// TIA Portal V20 export
FUNCTION_BLOCK "System_To_Moving_Pallets"   // FB15, LAD
{ S7_Optimized_Access := 'TRUE' }
// stored: MemoryReserve 100, SetENOAutomatically false
   VAR
      iCenterTippler : Bool;
      oCeterTippler : Bool;
      Reset_Centering_Tippler : Bool;
      ST13_ST14 { S7_SetPoint := 'True'} : "Pallet_Transport_Row_4";
      ST12_ST13 { S7_SetPoint := 'True'} : "Pallet_Transport_Row_4";
      ST11_ST12 { S7_SetPoint := 'True'} : "Pallet_Transport_Row_4";
      ST10_ST11 { S7_SetPoint := 'True'} : "Pallet_Transport_Row_4";
      ST09_ST10 { S7_SetPoint := 'True'} : "Pallet_Transport_Row_4";
      ST08_ST09 { S7_SetPoint := 'True'} : "Pallet_Transport_Row_4";
      ST07_ST08 { S7_SetPoint := 'True'} : "Pallet_Transport_Row_4";
      ST06_ST07 { S7_SetPoint := 'True'} : "Pallet_Transport_Row_4";
      ST05_ST06 { S7_SetPoint := 'True'} : "Pallet_Transport_Row_4";
      ST04_ST05 { S7_SetPoint := 'True'} : "Pallet_Transport_Row_4";
      ST01_ST02 { S7_SetPoint := 'True'} : "Pallet_Transport_Row_1_2";
      ST02_ST01 { S7_SetPoint := 'True'} : "Pallet_Transport_Row_1_2";
      ST38_ST01 { S7_SetPoint := 'True'} : "Pallet_Transport_Row_1_2";
      ST01_ST38 { S7_SetPoint := 'True'} : "Pallet_Transport_Row_1_2";
      ST34_ST35 { S7_SetPoint := 'True'} : "Pallet_Transport_Row_1_2";
      ST35_ST34 { S7_SetPoint := 'True'} : "Pallet_Transport_Row_1_2";
      ST33_ST34 { S7_SetPoint := 'True'} : "Pallet_Transport_Row_1_2";
      ST34_ST33 { S7_SetPoint := 'True'} : "Pallet_Transport_Row_1_2";
      ST32_ST33 { S7_SetPoint := 'True'} : "Pallet_Transport_Row_1_2";
      ST36_ST38 { S7_SetPoint := 'True'} : "Pallet_Transport_Row_1_2";
      ST38_ST36 { S7_SetPoint := 'True'} : "Pallet_Transport_Row_1_2";
      ST37_ST36 { S7_SetPoint := 'True'} : "Pallet_Transport_Row_1_2";
      ST18_ST37 { S7_SetPoint := 'True'} : "Pallet_Transport_Row_1_2";
      ST19_ST18 { S7_SetPoint := 'True'} : "Pallet_Transport_Row_1_2";
      ST20_ST19 { S7_SetPoint := 'True'} : "Pallet_Transport_Row_1_2";
      ST21_ST20 { S7_SetPoint := 'True'} : "Pallet_Transport_Row_1_2";
      ST22_ST21 { S7_SetPoint := 'True'} : "Pallet_Transport_Row_1_2";
      ST23_ST22 { S7_SetPoint := 'True'} : "Pallet_Transport_Row_1_2";
      ST24_ST23 { S7_SetPoint := 'True'} : "Pallet_Transport_Row_1_2";
      Centering_Perform : Array[7..13, 1..3] of Bool;
      Centering_Status { S7_SetPoint := 'True'} : Array[7..13, 1..3] of Bool;
      ST31_ST32 { S7_SetPoint := 'True'} : "Pallet_Transport_Row_1_2";
      ST30_ST31 { S7_SetPoint := 'True'} : "Pallet_Transport_Row_1_2";
      ST29_ST30 { S7_SetPoint := 'True'} : "Pallet_Transport_Row_1_2";
      ST28_ST29 { S7_SetPoint := 'True'} : "Pallet_Transport_Row_1_2";
      TON_Reset_Drives { S7_SetPoint := 'True'} : TON_TIME;
      TP_Reset_Drives { S7_SetPoint := 'True'} : TP_TIME;
      Reset_Drives_Var { S7_SetPoint := 'True'} : Bool;
      ST27_ST28 { S7_SetPoint := 'True'} : "Pallet_Transport_Row_1_2";
      ST26_ST27 { S7_SetPoint := 'True'} : "Pallet_Transport_Row_1_2";
      ST25_ST26 { S7_SetPoint := 'True'} : "Pallet_Transport_Row_1_2";
      tComm_W1 { S7_SetPoint := 'True'} : TON_TIME;
      tComm_W2 { S7_SetPoint := 'True'} : TON_TIME;
      tComm_W4 { S7_SetPoint := 'True'} : TON_TIME;
   END_VAR
   VAR_TEMP
      i : Int;
   END_VAR
BEGIN

REGION Network 1: Initialisation of pallets status
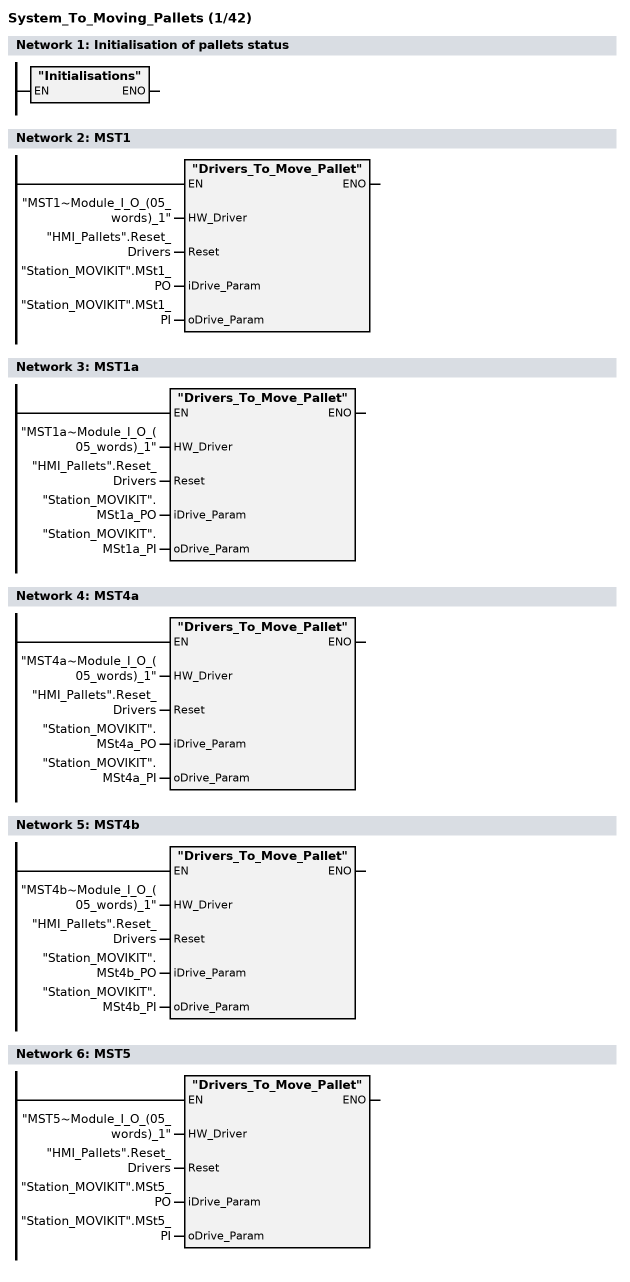
   RUNG wire#powerrail
      "Initialisations"()
   END_RUNG
   // the same network as SCL:
   "Initialisations"();
END_REGION

REGION Network 2: MST1
   RUNG wire#powerrail
      "Drivers_To_Move_Pallet"(HW_Driver := "MST1~Module_I_O_(05_words)_1", Reset := "HMI_Pallets".Reset_Drivers, iDrive_Param := "Station_MOVIKIT".MSt1_PO, oDrive_Param := "Station_MOVIKIT".MSt1_PI)
   END_RUNG
   // the same network as SCL:
   "Drivers_To_Move_Pallet"(HW_Driver := "MST1~Module_I_O_(05_words)_1",
                           Reset := "HMI_Pallets".Reset_Drivers,
                           iDrive_Param := "Station_MOVIKIT".MSt1_PO,
                           oDrive_Param := "Station_MOVIKIT".MSt1_PI);
END_REGION

REGION Network 3: MST1a
   RUNG wire#powerrail
      "Drivers_To_Move_Pallet"(HW_Driver := "MST1a~Module_I_O_(05_words)_1", Reset := "HMI_Pallets".Reset_Drivers, iDrive_Param := "Station_MOVIKIT".MSt1a_PO, oDrive_Param := "Station_MOVIKIT".MSt1a_PI)
   END_RUNG
   // the same network as SCL:
   "Drivers_To_Move_Pallet"(HW_Driver := "MST1a~Module_I_O_(05_words)_1",
                           Reset := "HMI_Pallets".Reset_Drivers,
                           iDrive_Param := "Station_MOVIKIT".MSt1a_PO,
                           oDrive_Param := "Station_MOVIKIT".MSt1a_PI);
END_REGION

REGION Network 4: MST4a
   RUNG wire#powerrail
      "Drivers_To_Move_Pallet"(HW_Driver := "MST4a~Module_I_O_(05_words)_1", Reset := "HMI_Pallets".Reset_Drivers, iDrive_Param := "Station_MOVIKIT".MSt4a_PO, oDrive_Param := "Station_MOVIKIT".MSt4a_PI)
   END_RUNG
   // the same network as SCL:
   "Drivers_To_Move_Pallet"(HW_Driver := "MST4a~Module_I_O_(05_words)_1",
                           Reset := "HMI_Pallets".Reset_Drivers,
                           iDrive_Param := "Station_MOVIKIT".MSt4a_PO,
                           oDrive_Param := "Station_MOVIKIT".MSt4a_PI);
END_REGION

REGION Network 5: MST4b
   RUNG wire#powerrail
      "Drivers_To_Move_Pallet"(HW_Driver := "MST4b~Module_I_O_(05_words)_1", Reset := "HMI_Pallets".Reset_Drivers, iDrive_Param := "Station_MOVIKIT".MSt4b_PO, oDrive_Param := "Station_MOVIKIT".MSt4b_PI)
   END_RUNG
   // the same network as SCL:
   "Drivers_To_Move_Pallet"(HW_Driver := "MST4b~Module_I_O_(05_words)_1",
                           Reset := "HMI_Pallets".Reset_Drivers,
                           iDrive_Param := "Station_MOVIKIT".MSt4b_PO,
                           oDrive_Param := "Station_MOVIKIT".MSt4b_PI);
END_REGION

REGION Network 6: MST5
   RUNG wire#powerrail
      "Drivers_To_Move_Pallet"(HW_Driver := "MST5~Module_I_O_(05_words)_1", Reset := "HMI_Pallets".Reset_Drivers, iDrive_Param := "Station_MOVIKIT".MSt5_PO, oDrive_Param := "Station_MOVIKIT".MSt5_PI)
   END_RUNG
   // the same network as SCL:
   "Drivers_To_Move_Pallet"(HW_Driver := "MST5~Module_I_O_(05_words)_1",
                           Reset := "HMI_Pallets".Reset_Drivers,
                           iDrive_Param := "Station_MOVIKIT".MSt5_PO,
                           oDrive_Param := "Station_MOVIKIT".MSt5_PI);
END_REGION

REGION Network 7: MST6a
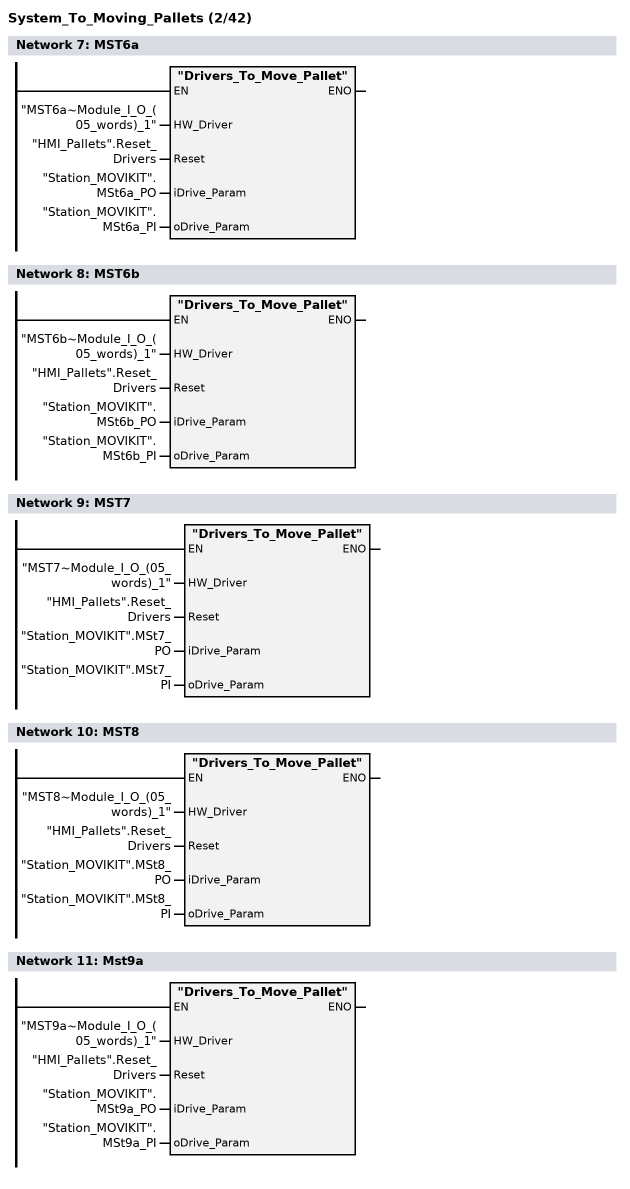
   RUNG wire#powerrail
      "Drivers_To_Move_Pallet"(HW_Driver := "MST6a~Module_I_O_(05_words)_1", Reset := "HMI_Pallets".Reset_Drivers, iDrive_Param := "Station_MOVIKIT".MSt6a_PO, oDrive_Param := "Station_MOVIKIT".MSt6a_PI)
   END_RUNG
   // the same network as SCL:
   "Drivers_To_Move_Pallet"(HW_Driver := "MST6a~Module_I_O_(05_words)_1",
                           Reset := "HMI_Pallets".Reset_Drivers,
                           iDrive_Param := "Station_MOVIKIT".MSt6a_PO,
                           oDrive_Param := "Station_MOVIKIT".MSt6a_PI);
END_REGION

REGION Network 8: MST6b
   RUNG wire#powerrail
      "Drivers_To_Move_Pallet"(HW_Driver := "MST6b~Module_I_O_(05_words)_1", Reset := "HMI_Pallets".Reset_Drivers, iDrive_Param := "Station_MOVIKIT".MSt6b_PO, oDrive_Param := "Station_MOVIKIT".MSt6b_PI)
   END_RUNG
   // the same network as SCL:
   "Drivers_To_Move_Pallet"(HW_Driver := "MST6b~Module_I_O_(05_words)_1",
                           Reset := "HMI_Pallets".Reset_Drivers,
                           iDrive_Param := "Station_MOVIKIT".MSt6b_PO,
                           oDrive_Param := "Station_MOVIKIT".MSt6b_PI);
END_REGION

REGION Network 9: MST7
   RUNG wire#powerrail
      "Drivers_To_Move_Pallet"(HW_Driver := "MST7~Module_I_O_(05_words)_1", Reset := "HMI_Pallets".Reset_Drivers, iDrive_Param := "Station_MOVIKIT".MSt7_PO, oDrive_Param := "Station_MOVIKIT".MSt7_PI)
   END_RUNG
   // the same network as SCL:
   "Drivers_To_Move_Pallet"(HW_Driver := "MST7~Module_I_O_(05_words)_1",
                           Reset := "HMI_Pallets".Reset_Drivers,
                           iDrive_Param := "Station_MOVIKIT".MSt7_PO,
                           oDrive_Param := "Station_MOVIKIT".MSt7_PI);
END_REGION

REGION Network 10: MST8
   RUNG wire#powerrail
      "Drivers_To_Move_Pallet"(HW_Driver := "MST8~Module_I_O_(05_words)_1", Reset := "HMI_Pallets".Reset_Drivers, iDrive_Param := "Station_MOVIKIT".MSt8_PO, oDrive_Param := "Station_MOVIKIT".MSt8_PI)
   END_RUNG
   // the same network as SCL:
   "Drivers_To_Move_Pallet"(HW_Driver := "MST8~Module_I_O_(05_words)_1",
                           Reset := "HMI_Pallets".Reset_Drivers,
                           iDrive_Param := "Station_MOVIKIT".MSt8_PO,
                           oDrive_Param := "Station_MOVIKIT".MSt8_PI);
END_REGION

REGION Network 11: Mst9a
   RUNG wire#powerrail
      "Drivers_To_Move_Pallet"(HW_Driver := "MST9a~Module_I_O_(05_words)_1", Reset := "HMI_Pallets".Reset_Drivers, iDrive_Param := "Station_MOVIKIT".MSt9a_PO, oDrive_Param := "Station_MOVIKIT".MSt9a_PI)
   END_RUNG
   // the same network as SCL:
   "Drivers_To_Move_Pallet"(HW_Driver := "MST9a~Module_I_O_(05_words)_1",
                           Reset := "HMI_Pallets".Reset_Drivers,
                           iDrive_Param := "Station_MOVIKIT".MSt9a_PO,
                           oDrive_Param := "Station_MOVIKIT".MSt9a_PI);
END_REGION

REGION Network 12: Mst9b
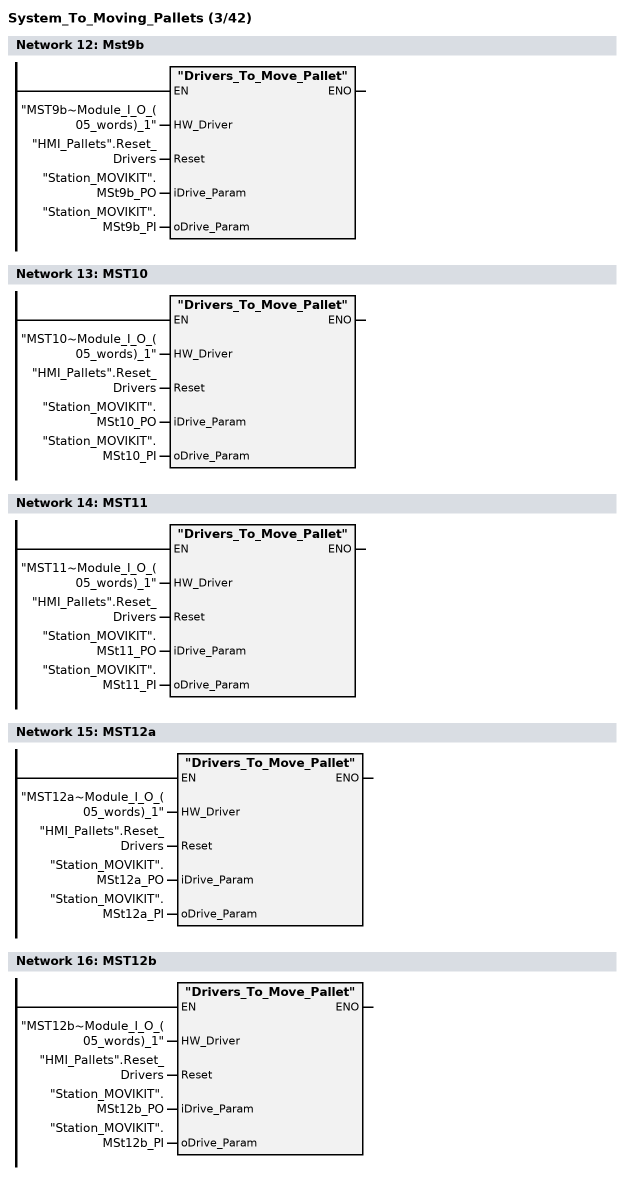
   RUNG wire#powerrail
      "Drivers_To_Move_Pallet"(HW_Driver := "MST9b~Module_I_O_(05_words)_1", Reset := "HMI_Pallets".Reset_Drivers, iDrive_Param := "Station_MOVIKIT".MSt9b_PO, oDrive_Param := "Station_MOVIKIT".MSt9b_PI)
   END_RUNG
   // the same network as SCL:
   "Drivers_To_Move_Pallet"(HW_Driver := "MST9b~Module_I_O_(05_words)_1",
                           Reset := "HMI_Pallets".Reset_Drivers,
                           iDrive_Param := "Station_MOVIKIT".MSt9b_PO,
                           oDrive_Param := "Station_MOVIKIT".MSt9b_PI);
END_REGION

REGION Network 13: MST10
   RUNG wire#powerrail
      "Drivers_To_Move_Pallet"(HW_Driver := "MST10~Module_I_O_(05_words)_1", Reset := "HMI_Pallets".Reset_Drivers, iDrive_Param := "Station_MOVIKIT".MSt10_PO, oDrive_Param := "Station_MOVIKIT".MSt10_PI)
   END_RUNG
   // the same network as SCL:
   "Drivers_To_Move_Pallet"(HW_Driver := "MST10~Module_I_O_(05_words)_1",
                           Reset := "HMI_Pallets".Reset_Drivers,
                           iDrive_Param := "Station_MOVIKIT".MSt10_PO,
                           oDrive_Param := "Station_MOVIKIT".MSt10_PI);
END_REGION

REGION Network 14: MST11
   RUNG wire#powerrail
      "Drivers_To_Move_Pallet"(HW_Driver := "MST11~Module_I_O_(05_words)_1", Reset := "HMI_Pallets".Reset_Drivers, iDrive_Param := "Station_MOVIKIT".MSt11_PO, oDrive_Param := "Station_MOVIKIT".MSt11_PI)
   END_RUNG
   // the same network as SCL:
   "Drivers_To_Move_Pallet"(HW_Driver := "MST11~Module_I_O_(05_words)_1",
                           Reset := "HMI_Pallets".Reset_Drivers,
                           iDrive_Param := "Station_MOVIKIT".MSt11_PO,
                           oDrive_Param := "Station_MOVIKIT".MSt11_PI);
END_REGION

REGION Network 15: MST12a
   RUNG wire#powerrail
      "Drivers_To_Move_Pallet"(HW_Driver := "MST12a~Module_I_O_(05_words)_1", Reset := "HMI_Pallets".Reset_Drivers, iDrive_Param := "Station_MOVIKIT".MSt12a_PO, oDrive_Param := "Station_MOVIKIT".MSt12a_PI)
   END_RUNG
   // the same network as SCL:
   "Drivers_To_Move_Pallet"(HW_Driver := "MST12a~Module_I_O_(05_words)_1",
                           Reset := "HMI_Pallets".Reset_Drivers,
                           iDrive_Param := "Station_MOVIKIT".MSt12a_PO,
                           oDrive_Param := "Station_MOVIKIT".MSt12a_PI);
END_REGION

REGION Network 16: MST12b
   RUNG wire#powerrail
      "Drivers_To_Move_Pallet"(HW_Driver := "MST12b~Module_I_O_(05_words)_1", Reset := "HMI_Pallets".Reset_Drivers, iDrive_Param := "Station_MOVIKIT".MSt12b_PO, oDrive_Param := "Station_MOVIKIT".MSt12b_PI)
   END_RUNG
   // the same network as SCL:
   "Drivers_To_Move_Pallet"(HW_Driver := "MST12b~Module_I_O_(05_words)_1",
                           Reset := "HMI_Pallets".Reset_Drivers,
                           iDrive_Param := "Station_MOVIKIT".MSt12b_PO,
                           oDrive_Param := "Station_MOVIKIT".MSt12b_PI);
END_REGION

REGION Network 17: MST13
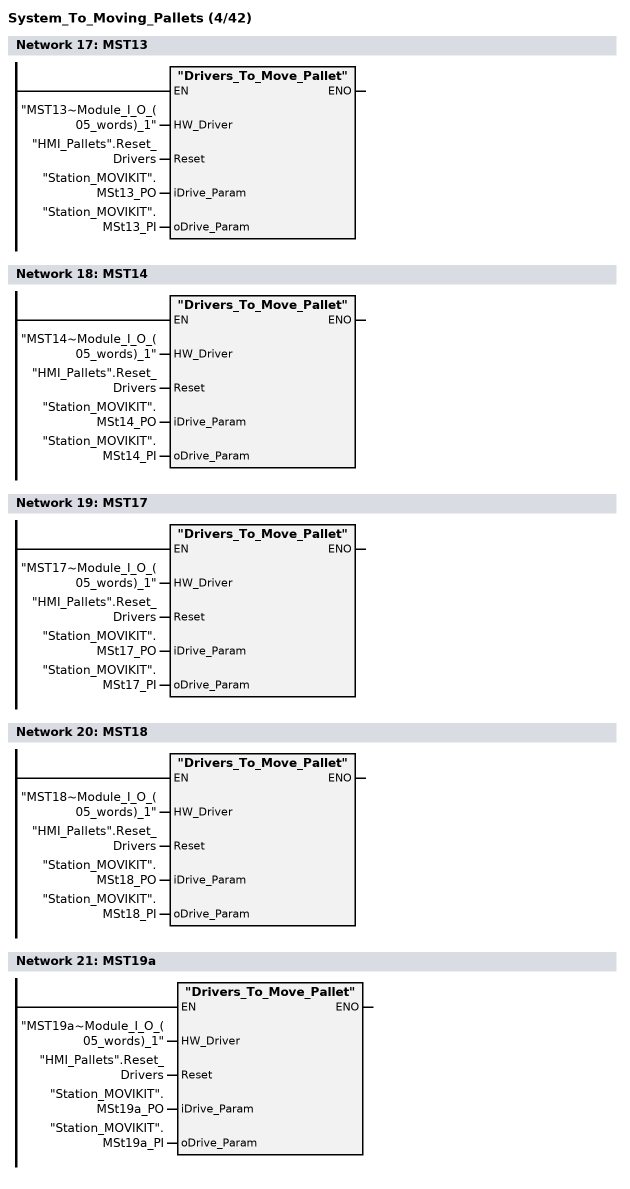
   RUNG wire#powerrail
      "Drivers_To_Move_Pallet"(HW_Driver := "MST13~Module_I_O_(05_words)_1", Reset := "HMI_Pallets".Reset_Drivers, iDrive_Param := "Station_MOVIKIT".MSt13_PO, oDrive_Param := "Station_MOVIKIT".MSt13_PI)
   END_RUNG
   // the same network as SCL:
   "Drivers_To_Move_Pallet"(HW_Driver := "MST13~Module_I_O_(05_words)_1",
                           Reset := "HMI_Pallets".Reset_Drivers,
                           iDrive_Param := "Station_MOVIKIT".MSt13_PO,
                           oDrive_Param := "Station_MOVIKIT".MSt13_PI);
END_REGION

REGION Network 18: MST14
   RUNG wire#powerrail
      "Drivers_To_Move_Pallet"(HW_Driver := "MST14~Module_I_O_(05_words)_1", Reset := "HMI_Pallets".Reset_Drivers, iDrive_Param := "Station_MOVIKIT".MSt14_PO, oDrive_Param := "Station_MOVIKIT".MSt14_PI)
   END_RUNG
   // the same network as SCL:
   "Drivers_To_Move_Pallet"(HW_Driver := "MST14~Module_I_O_(05_words)_1",
                           Reset := "HMI_Pallets".Reset_Drivers,
                           iDrive_Param := "Station_MOVIKIT".MSt14_PO,
                           oDrive_Param := "Station_MOVIKIT".MSt14_PI);
END_REGION

REGION Network 19: MST17
   RUNG wire#powerrail
      "Drivers_To_Move_Pallet"(HW_Driver := "MST17~Module_I_O_(05_words)_1", Reset := "HMI_Pallets".Reset_Drivers, iDrive_Param := "Station_MOVIKIT".MSt17_PO, oDrive_Param := "Station_MOVIKIT".MSt17_PI)
   END_RUNG
   // the same network as SCL:
   "Drivers_To_Move_Pallet"(HW_Driver := "MST17~Module_I_O_(05_words)_1",
                           Reset := "HMI_Pallets".Reset_Drivers,
                           iDrive_Param := "Station_MOVIKIT".MSt17_PO,
                           oDrive_Param := "Station_MOVIKIT".MSt17_PI);
END_REGION

REGION Network 20: MST18
   RUNG wire#powerrail
      "Drivers_To_Move_Pallet"(HW_Driver := "MST18~Module_I_O_(05_words)_1", Reset := "HMI_Pallets".Reset_Drivers, iDrive_Param := "Station_MOVIKIT".MSt18_PO, oDrive_Param := "Station_MOVIKIT".MSt18_PI)
   END_RUNG
   // the same network as SCL:
   "Drivers_To_Move_Pallet"(HW_Driver := "MST18~Module_I_O_(05_words)_1",
                           Reset := "HMI_Pallets".Reset_Drivers,
                           iDrive_Param := "Station_MOVIKIT".MSt18_PO,
                           oDrive_Param := "Station_MOVIKIT".MSt18_PI);
END_REGION

REGION Network 21: MST19a
   RUNG wire#powerrail
      "Drivers_To_Move_Pallet"(HW_Driver := "MST19a~Module_I_O_(05_words)_1", Reset := "HMI_Pallets".Reset_Drivers, iDrive_Param := "Station_MOVIKIT".MSt19a_PO, oDrive_Param := "Station_MOVIKIT".MSt19a_PI)
   END_RUNG
   // the same network as SCL:
   "Drivers_To_Move_Pallet"(HW_Driver := "MST19a~Module_I_O_(05_words)_1",
                           Reset := "HMI_Pallets".Reset_Drivers,
                           iDrive_Param := "Station_MOVIKIT".MSt19a_PO,
                           oDrive_Param := "Station_MOVIKIT".MSt19a_PI);
END_REGION

REGION Network 22: MST19b
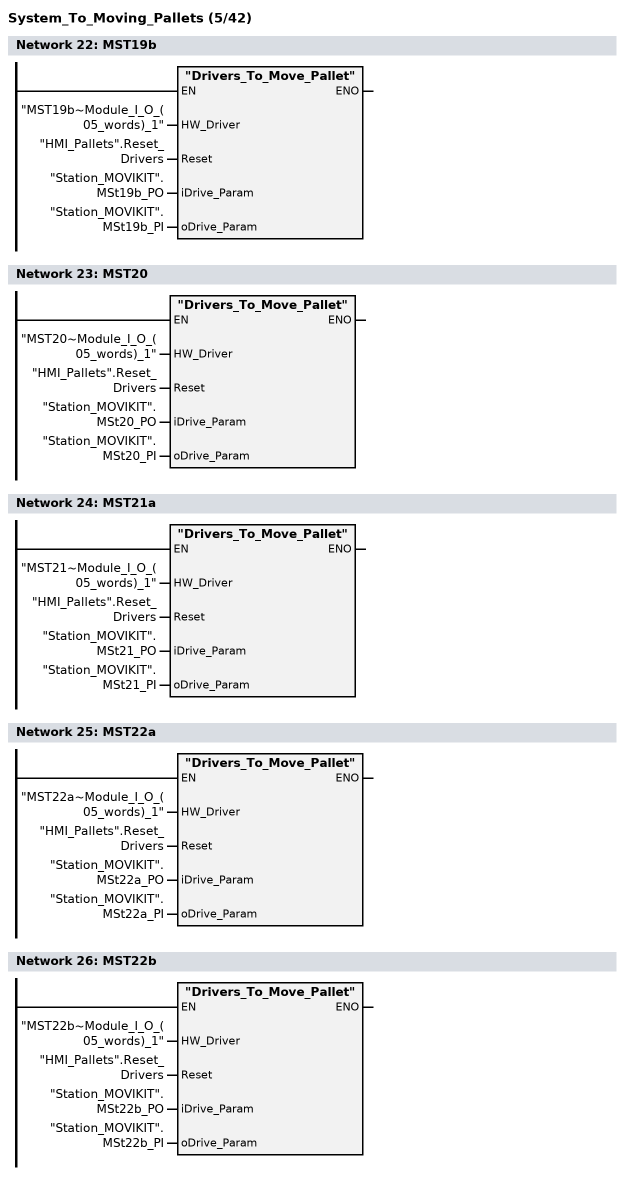
   RUNG wire#powerrail
      "Drivers_To_Move_Pallet"(HW_Driver := "MST19b~Module_I_O_(05_words)_1", Reset := "HMI_Pallets".Reset_Drivers, iDrive_Param := "Station_MOVIKIT".MSt19b_PO, oDrive_Param := "Station_MOVIKIT".MSt19b_PI)
   END_RUNG
   // the same network as SCL:
   "Drivers_To_Move_Pallet"(HW_Driver := "MST19b~Module_I_O_(05_words)_1",
                           Reset := "HMI_Pallets".Reset_Drivers,
                           iDrive_Param := "Station_MOVIKIT".MSt19b_PO,
                           oDrive_Param := "Station_MOVIKIT".MSt19b_PI);
END_REGION

REGION Network 23: MST20
   RUNG wire#powerrail
      "Drivers_To_Move_Pallet"(HW_Driver := "MST20~Module_I_O_(05_words)_1", Reset := "HMI_Pallets".Reset_Drivers, iDrive_Param := "Station_MOVIKIT".MSt20_PO, oDrive_Param := "Station_MOVIKIT".MSt20_PI)
   END_RUNG
   // the same network as SCL:
   "Drivers_To_Move_Pallet"(HW_Driver := "MST20~Module_I_O_(05_words)_1",
                           Reset := "HMI_Pallets".Reset_Drivers,
                           iDrive_Param := "Station_MOVIKIT".MSt20_PO,
                           oDrive_Param := "Station_MOVIKIT".MSt20_PI);
END_REGION

REGION Network 24: MST21a
   RUNG wire#powerrail
      "Drivers_To_Move_Pallet"(HW_Driver := "MST21~Module_I_O_(05_words)_1", Reset := "HMI_Pallets".Reset_Drivers, iDrive_Param := "Station_MOVIKIT".MSt21_PO, oDrive_Param := "Station_MOVIKIT".MSt21_PI)
   END_RUNG
   // the same network as SCL:
   "Drivers_To_Move_Pallet"(HW_Driver := "MST21~Module_I_O_(05_words)_1",
                           Reset := "HMI_Pallets".Reset_Drivers,
                           iDrive_Param := "Station_MOVIKIT".MSt21_PO,
                           oDrive_Param := "Station_MOVIKIT".MSt21_PI);
END_REGION

REGION Network 25: MST22a
   RUNG wire#powerrail
      "Drivers_To_Move_Pallet"(HW_Driver := "MST22a~Module_I_O_(05_words)_1", Reset := "HMI_Pallets".Reset_Drivers, iDrive_Param := "Station_MOVIKIT".MSt22a_PO, oDrive_Param := "Station_MOVIKIT".MSt22a_PI)
   END_RUNG
   // the same network as SCL:
   "Drivers_To_Move_Pallet"(HW_Driver := "MST22a~Module_I_O_(05_words)_1",
                           Reset := "HMI_Pallets".Reset_Drivers,
                           iDrive_Param := "Station_MOVIKIT".MSt22a_PO,
                           oDrive_Param := "Station_MOVIKIT".MSt22a_PI);
END_REGION

REGION Network 26: MST22b
   RUNG wire#powerrail
      "Drivers_To_Move_Pallet"(HW_Driver := "MST22b~Module_I_O_(05_words)_1", Reset := "HMI_Pallets".Reset_Drivers, iDrive_Param := "Station_MOVIKIT".MSt22b_PO, oDrive_Param := "Station_MOVIKIT".MSt22b_PI)
   END_RUNG
   // the same network as SCL:
   "Drivers_To_Move_Pallet"(HW_Driver := "MST22b~Module_I_O_(05_words)_1",
                           Reset := "HMI_Pallets".Reset_Drivers,
                           iDrive_Param := "Station_MOVIKIT".MSt22b_PO,
                           oDrive_Param := "Station_MOVIKIT".MSt22b_PI);
END_REGION

REGION Network 27: MST23a
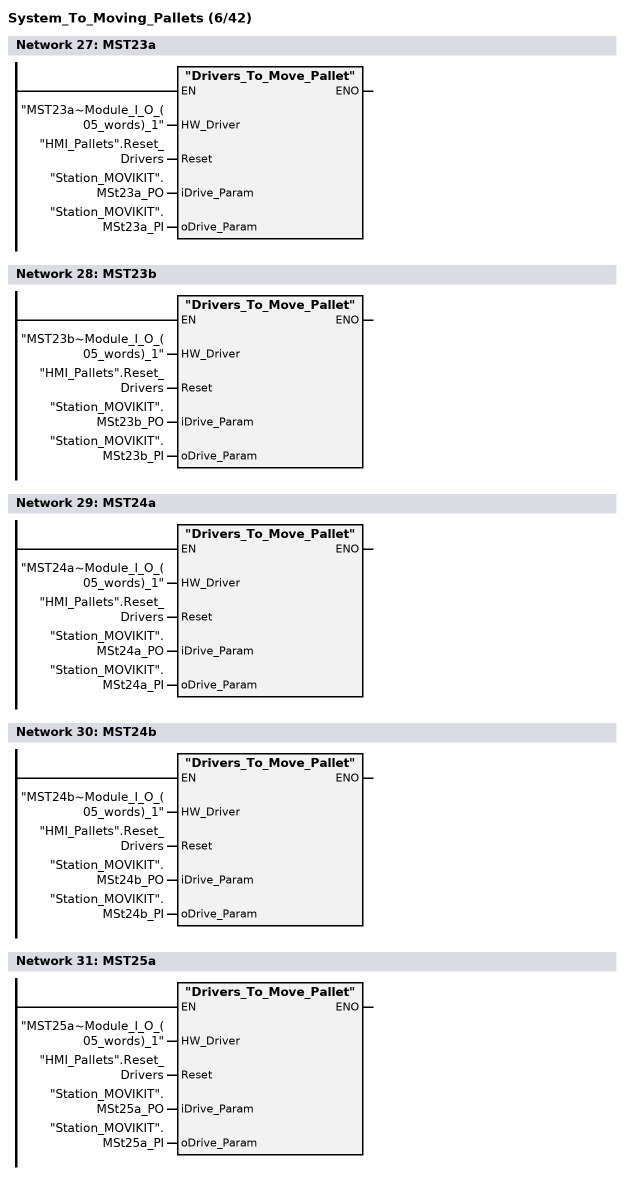
   RUNG wire#powerrail
      "Drivers_To_Move_Pallet"(HW_Driver := "MST23a~Module_I_O_(05_words)_1", Reset := "HMI_Pallets".Reset_Drivers, iDrive_Param := "Station_MOVIKIT".MSt23a_PO, oDrive_Param := "Station_MOVIKIT".MSt23a_PI)
   END_RUNG
   // the same network as SCL:
   "Drivers_To_Move_Pallet"(HW_Driver := "MST23a~Module_I_O_(05_words)_1",
                           Reset := "HMI_Pallets".Reset_Drivers,
                           iDrive_Param := "Station_MOVIKIT".MSt23a_PO,
                           oDrive_Param := "Station_MOVIKIT".MSt23a_PI);
END_REGION

REGION Network 28: MST23b
   RUNG wire#powerrail
      "Drivers_To_Move_Pallet"(HW_Driver := "MST23b~Module_I_O_(05_words)_1", Reset := "HMI_Pallets".Reset_Drivers, iDrive_Param := "Station_MOVIKIT".MSt23b_PO, oDrive_Param := "Station_MOVIKIT".MSt23b_PI)
   END_RUNG
   // the same network as SCL:
   "Drivers_To_Move_Pallet"(HW_Driver := "MST23b~Module_I_O_(05_words)_1",
                           Reset := "HMI_Pallets".Reset_Drivers,
                           iDrive_Param := "Station_MOVIKIT".MSt23b_PO,
                           oDrive_Param := "Station_MOVIKIT".MSt23b_PI);
END_REGION

REGION Network 29: MST24a
   RUNG wire#powerrail
      "Drivers_To_Move_Pallet"(HW_Driver := "MST24a~Module_I_O_(05_words)_1", Reset := "HMI_Pallets".Reset_Drivers, iDrive_Param := "Station_MOVIKIT".MSt24a_PO, oDrive_Param := "Station_MOVIKIT".MSt24a_PI)
   END_RUNG
   // the same network as SCL:
   "Drivers_To_Move_Pallet"(HW_Driver := "MST24a~Module_I_O_(05_words)_1",
                           Reset := "HMI_Pallets".Reset_Drivers,
                           iDrive_Param := "Station_MOVIKIT".MSt24a_PO,
                           oDrive_Param := "Station_MOVIKIT".MSt24a_PI);
END_REGION

REGION Network 30: MST24b
   RUNG wire#powerrail
      "Drivers_To_Move_Pallet"(HW_Driver := "MST24b~Module_I_O_(05_words)_1", Reset := "HMI_Pallets".Reset_Drivers, iDrive_Param := "Station_MOVIKIT".MSt24b_PO, oDrive_Param := "Station_MOVIKIT".MSt24b_PI)
   END_RUNG
   // the same network as SCL:
   "Drivers_To_Move_Pallet"(HW_Driver := "MST24b~Module_I_O_(05_words)_1",
                           Reset := "HMI_Pallets".Reset_Drivers,
                           iDrive_Param := "Station_MOVIKIT".MSt24b_PO,
                           oDrive_Param := "Station_MOVIKIT".MSt24b_PI);
END_REGION

REGION Network 31: MST25a
   RUNG wire#powerrail
      "Drivers_To_Move_Pallet"(HW_Driver := "MST25a~Module_I_O_(05_words)_1", Reset := "HMI_Pallets".Reset_Drivers, iDrive_Param := "Station_MOVIKIT".MSt25a_PO, oDrive_Param := "Station_MOVIKIT".MSt25a_PI)
   END_RUNG
   // the same network as SCL:
   "Drivers_To_Move_Pallet"(HW_Driver := "MST25a~Module_I_O_(05_words)_1",
                           Reset := "HMI_Pallets".Reset_Drivers,
                           iDrive_Param := "Station_MOVIKIT".MSt25a_PO,
                           oDrive_Param := "Station_MOVIKIT".MSt25a_PI);
END_REGION

REGION Network 32: MST25b
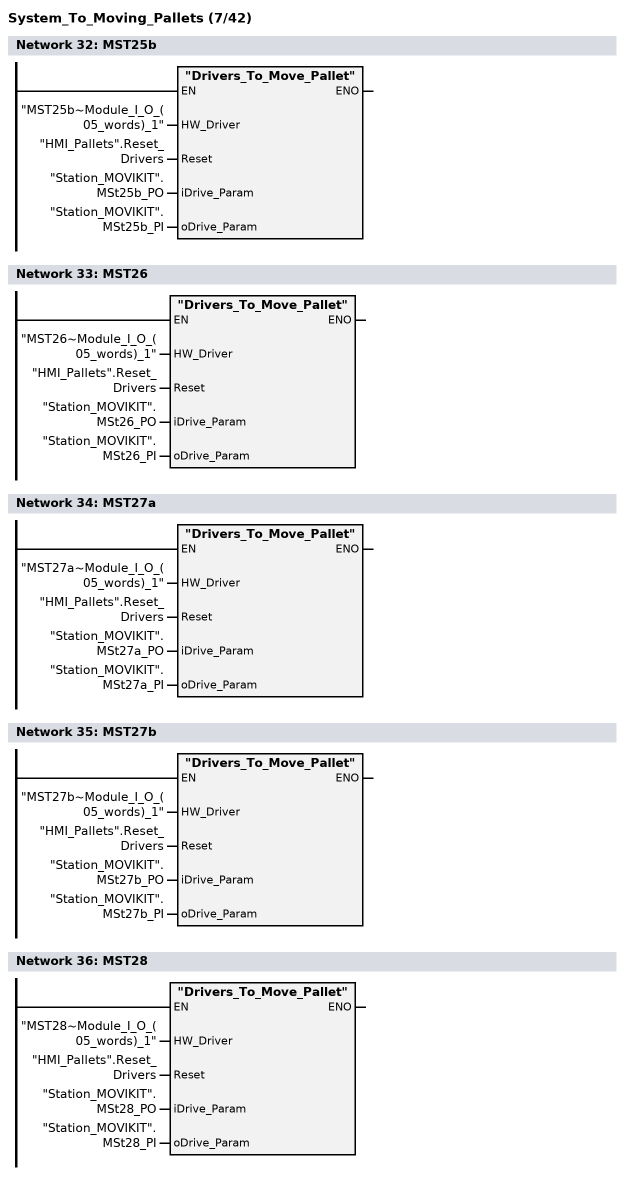
   RUNG wire#powerrail
      "Drivers_To_Move_Pallet"(HW_Driver := "MST25b~Module_I_O_(05_words)_1", Reset := "HMI_Pallets".Reset_Drivers, iDrive_Param := "Station_MOVIKIT".MSt25b_PO, oDrive_Param := "Station_MOVIKIT".MSt25b_PI)
   END_RUNG
   // the same network as SCL:
   "Drivers_To_Move_Pallet"(HW_Driver := "MST25b~Module_I_O_(05_words)_1",
                           Reset := "HMI_Pallets".Reset_Drivers,
                           iDrive_Param := "Station_MOVIKIT".MSt25b_PO,
                           oDrive_Param := "Station_MOVIKIT".MSt25b_PI);
END_REGION

REGION Network 33: MST26
   RUNG wire#powerrail
      "Drivers_To_Move_Pallet"(HW_Driver := "MST26~Module_I_O_(05_words)_1", Reset := "HMI_Pallets".Reset_Drivers, iDrive_Param := "Station_MOVIKIT".MSt26_PO, oDrive_Param := "Station_MOVIKIT".MSt26_PI)
   END_RUNG
   // the same network as SCL:
   "Drivers_To_Move_Pallet"(HW_Driver := "MST26~Module_I_O_(05_words)_1",
                           Reset := "HMI_Pallets".Reset_Drivers,
                           iDrive_Param := "Station_MOVIKIT".MSt26_PO,
                           oDrive_Param := "Station_MOVIKIT".MSt26_PI);
END_REGION

REGION Network 34: MST27a
   RUNG wire#powerrail
      "Drivers_To_Move_Pallet"(HW_Driver := "MST27a~Module_I_O_(05_words)_1", Reset := "HMI_Pallets".Reset_Drivers, iDrive_Param := "Station_MOVIKIT".MSt27a_PO, oDrive_Param := "Station_MOVIKIT".MSt27a_PI)
   END_RUNG
   // the same network as SCL:
   "Drivers_To_Move_Pallet"(HW_Driver := "MST27a~Module_I_O_(05_words)_1",
                           Reset := "HMI_Pallets".Reset_Drivers,
                           iDrive_Param := "Station_MOVIKIT".MSt27a_PO,
                           oDrive_Param := "Station_MOVIKIT".MSt27a_PI);
END_REGION

REGION Network 35: MST27b
   RUNG wire#powerrail
      "Drivers_To_Move_Pallet"(HW_Driver := "MST27b~Module_I_O_(05_words)_1", Reset := "HMI_Pallets".Reset_Drivers, iDrive_Param := "Station_MOVIKIT".MSt27b_PO, oDrive_Param := "Station_MOVIKIT".MSt27b_PI)
   END_RUNG
   // the same network as SCL:
   "Drivers_To_Move_Pallet"(HW_Driver := "MST27b~Module_I_O_(05_words)_1",
                           Reset := "HMI_Pallets".Reset_Drivers,
                           iDrive_Param := "Station_MOVIKIT".MSt27b_PO,
                           oDrive_Param := "Station_MOVIKIT".MSt27b_PI);
END_REGION

REGION Network 36: MST28
   RUNG wire#powerrail
      "Drivers_To_Move_Pallet"(HW_Driver := "MST28~Module_I_O_(05_words)_1", Reset := "HMI_Pallets".Reset_Drivers, iDrive_Param := "Station_MOVIKIT".MSt28_PO, oDrive_Param := "Station_MOVIKIT".MSt28_PI)
   END_RUNG
   // the same network as SCL:
   "Drivers_To_Move_Pallet"(HW_Driver := "MST28~Module_I_O_(05_words)_1",
                           Reset := "HMI_Pallets".Reset_Drivers,
                           iDrive_Param := "Station_MOVIKIT".MSt28_PO,
                           oDrive_Param := "Station_MOVIKIT".MSt28_PI);
END_REGION

REGION Network 37: MST29
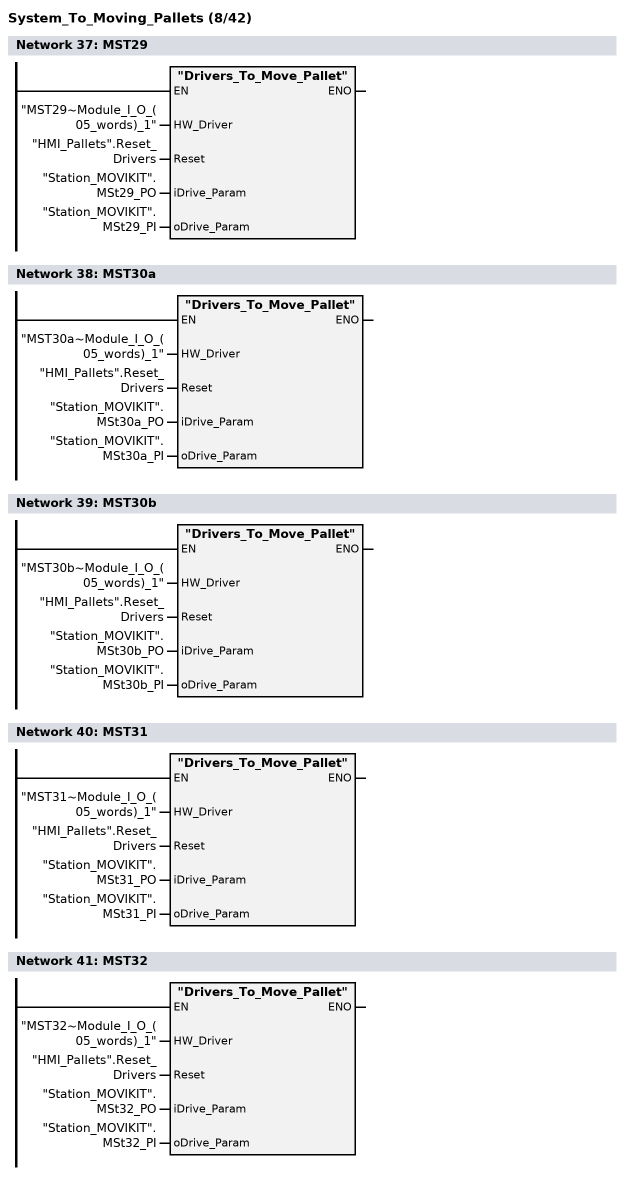
   RUNG wire#powerrail
      "Drivers_To_Move_Pallet"(HW_Driver := "MST29~Module_I_O_(05_words)_1", Reset := "HMI_Pallets".Reset_Drivers, iDrive_Param := "Station_MOVIKIT".MSt29_PO, oDrive_Param := "Station_MOVIKIT".MSt29_PI)
   END_RUNG
   // the same network as SCL:
   "Drivers_To_Move_Pallet"(HW_Driver := "MST29~Module_I_O_(05_words)_1",
                           Reset := "HMI_Pallets".Reset_Drivers,
                           iDrive_Param := "Station_MOVIKIT".MSt29_PO,
                           oDrive_Param := "Station_MOVIKIT".MSt29_PI);
END_REGION

REGION Network 38: MST30a
   RUNG wire#powerrail
      "Drivers_To_Move_Pallet"(HW_Driver := "MST30a~Module_I_O_(05_words)_1", Reset := "HMI_Pallets".Reset_Drivers, iDrive_Param := "Station_MOVIKIT".MSt30a_PO, oDrive_Param := "Station_MOVIKIT".MSt30a_PI)
   END_RUNG
   // the same network as SCL:
   "Drivers_To_Move_Pallet"(HW_Driver := "MST30a~Module_I_O_(05_words)_1",
                           Reset := "HMI_Pallets".Reset_Drivers,
                           iDrive_Param := "Station_MOVIKIT".MSt30a_PO,
                           oDrive_Param := "Station_MOVIKIT".MSt30a_PI);
END_REGION

REGION Network 39: MST30b
   RUNG wire#powerrail
      "Drivers_To_Move_Pallet"(HW_Driver := "MST30b~Module_I_O_(05_words)_1", Reset := "HMI_Pallets".Reset_Drivers, iDrive_Param := "Station_MOVIKIT".MSt30b_PO, oDrive_Param := "Station_MOVIKIT".MSt30b_PI)
   END_RUNG
   // the same network as SCL:
   "Drivers_To_Move_Pallet"(HW_Driver := "MST30b~Module_I_O_(05_words)_1",
                           Reset := "HMI_Pallets".Reset_Drivers,
                           iDrive_Param := "Station_MOVIKIT".MSt30b_PO,
                           oDrive_Param := "Station_MOVIKIT".MSt30b_PI);
END_REGION

REGION Network 40: MST31
   RUNG wire#powerrail
      "Drivers_To_Move_Pallet"(HW_Driver := "MST31~Module_I_O_(05_words)_1", Reset := "HMI_Pallets".Reset_Drivers, iDrive_Param := "Station_MOVIKIT".MSt31_PO, oDrive_Param := "Station_MOVIKIT".MSt31_PI)
   END_RUNG
   // the same network as SCL:
   "Drivers_To_Move_Pallet"(HW_Driver := "MST31~Module_I_O_(05_words)_1",
                           Reset := "HMI_Pallets".Reset_Drivers,
                           iDrive_Param := "Station_MOVIKIT".MSt31_PO,
                           oDrive_Param := "Station_MOVIKIT".MSt31_PI);
END_REGION

REGION Network 41: MST32
   RUNG wire#powerrail
      "Drivers_To_Move_Pallet"(HW_Driver := "MST32~Module_I_O_(05_words)_1", Reset := "HMI_Pallets".Reset_Drivers, iDrive_Param := "Station_MOVIKIT".MSt32_PO, oDrive_Param := "Station_MOVIKIT".MSt32_PI)
   END_RUNG
   // the same network as SCL:
   "Drivers_To_Move_Pallet"(HW_Driver := "MST32~Module_I_O_(05_words)_1",
                           Reset := "HMI_Pallets".Reset_Drivers,
                           iDrive_Param := "Station_MOVIKIT".MSt32_PO,
                           oDrive_Param := "Station_MOVIKIT".MSt32_PI);
END_REGION

REGION Network 42: MST33a
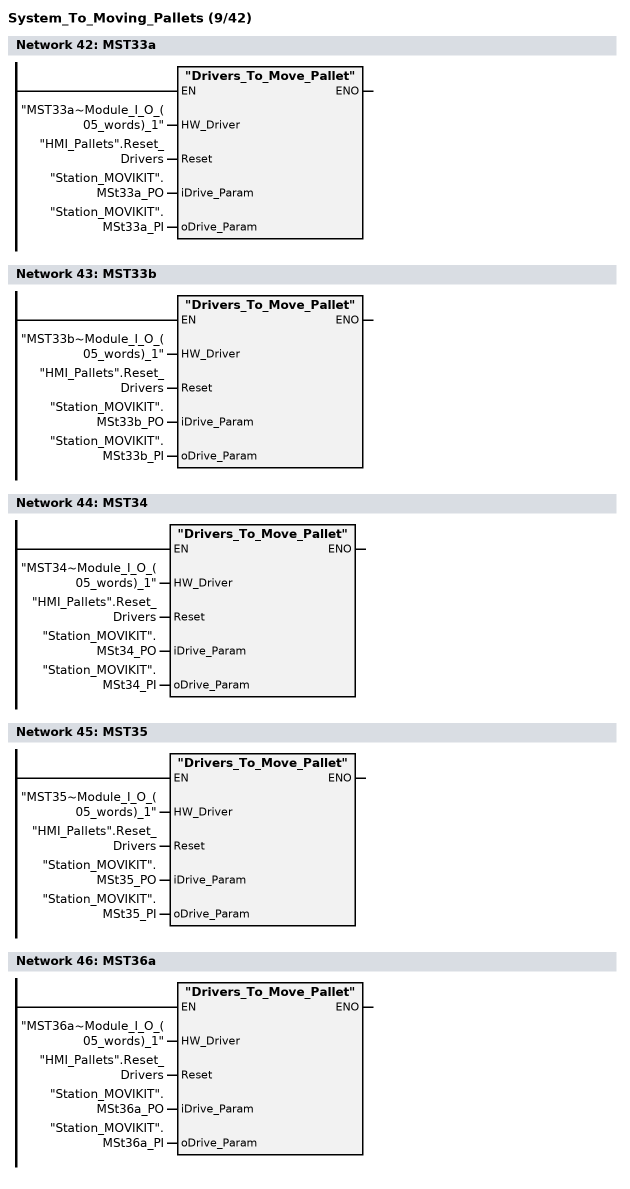
   RUNG wire#powerrail
      "Drivers_To_Move_Pallet"(HW_Driver := "MST33a~Module_I_O_(05_words)_1", Reset := "HMI_Pallets".Reset_Drivers, iDrive_Param := "Station_MOVIKIT".MSt33a_PO, oDrive_Param := "Station_MOVIKIT".MSt33a_PI)
   END_RUNG
   // the same network as SCL:
   "Drivers_To_Move_Pallet"(HW_Driver := "MST33a~Module_I_O_(05_words)_1",
                           Reset := "HMI_Pallets".Reset_Drivers,
                           iDrive_Param := "Station_MOVIKIT".MSt33a_PO,
                           oDrive_Param := "Station_MOVIKIT".MSt33a_PI);
END_REGION

REGION Network 43: MST33b
   RUNG wire#powerrail
      "Drivers_To_Move_Pallet"(HW_Driver := "MST33b~Module_I_O_(05_words)_1", Reset := "HMI_Pallets".Reset_Drivers, iDrive_Param := "Station_MOVIKIT".MSt33b_PO, oDrive_Param := "Station_MOVIKIT".MSt33b_PI)
   END_RUNG
   // the same network as SCL:
   "Drivers_To_Move_Pallet"(HW_Driver := "MST33b~Module_I_O_(05_words)_1",
                           Reset := "HMI_Pallets".Reset_Drivers,
                           iDrive_Param := "Station_MOVIKIT".MSt33b_PO,
                           oDrive_Param := "Station_MOVIKIT".MSt33b_PI);
END_REGION

REGION Network 44: MST34
   RUNG wire#powerrail
      "Drivers_To_Move_Pallet"(HW_Driver := "MST34~Module_I_O_(05_words)_1", Reset := "HMI_Pallets".Reset_Drivers, iDrive_Param := "Station_MOVIKIT".MSt34_PO, oDrive_Param := "Station_MOVIKIT".MSt34_PI)
   END_RUNG
   // the same network as SCL:
   "Drivers_To_Move_Pallet"(HW_Driver := "MST34~Module_I_O_(05_words)_1",
                           Reset := "HMI_Pallets".Reset_Drivers,
                           iDrive_Param := "Station_MOVIKIT".MSt34_PO,
                           oDrive_Param := "Station_MOVIKIT".MSt34_PI);
END_REGION

REGION Network 45: MST35
   RUNG wire#powerrail
      "Drivers_To_Move_Pallet"(HW_Driver := "MST35~Module_I_O_(05_words)_1", Reset := "HMI_Pallets".Reset_Drivers, iDrive_Param := "Station_MOVIKIT".MSt35_PO, oDrive_Param := "Station_MOVIKIT".MSt35_PI)
   END_RUNG
   // the same network as SCL:
   "Drivers_To_Move_Pallet"(HW_Driver := "MST35~Module_I_O_(05_words)_1",
                           Reset := "HMI_Pallets".Reset_Drivers,
                           iDrive_Param := "Station_MOVIKIT".MSt35_PO,
                           oDrive_Param := "Station_MOVIKIT".MSt35_PI);
END_REGION

REGION Network 46: MST36a
   RUNG wire#powerrail
      "Drivers_To_Move_Pallet"(HW_Driver := "MST36a~Module_I_O_(05_words)_1", Reset := "HMI_Pallets".Reset_Drivers, iDrive_Param := "Station_MOVIKIT".MSt36a_PO, oDrive_Param := "Station_MOVIKIT".MSt36a_PI)
   END_RUNG
   // the same network as SCL:
   "Drivers_To_Move_Pallet"(HW_Driver := "MST36a~Module_I_O_(05_words)_1",
                           Reset := "HMI_Pallets".Reset_Drivers,
                           iDrive_Param := "Station_MOVIKIT".MSt36a_PO,
                           oDrive_Param := "Station_MOVIKIT".MSt36a_PI);
END_REGION

REGION Network 47: MST36b
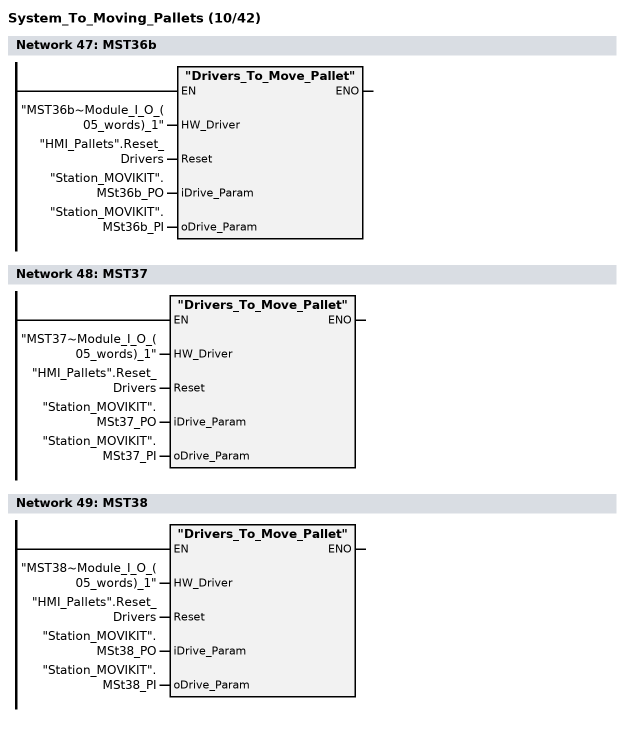
   RUNG wire#powerrail
      "Drivers_To_Move_Pallet"(HW_Driver := "MST36b~Module_I_O_(05_words)_1", Reset := "HMI_Pallets".Reset_Drivers, iDrive_Param := "Station_MOVIKIT".MSt36b_PO, oDrive_Param := "Station_MOVIKIT".MSt36b_PI)
   END_RUNG
   // the same network as SCL:
   "Drivers_To_Move_Pallet"(HW_Driver := "MST36b~Module_I_O_(05_words)_1",
                           Reset := "HMI_Pallets".Reset_Drivers,
                           iDrive_Param := "Station_MOVIKIT".MSt36b_PO,
                           oDrive_Param := "Station_MOVIKIT".MSt36b_PI);
END_REGION

REGION Network 48: MST37
   RUNG wire#powerrail
      "Drivers_To_Move_Pallet"(HW_Driver := "MST37~Module_I_O_(05_words)_1", Reset := "HMI_Pallets".Reset_Drivers, iDrive_Param := "Station_MOVIKIT".MSt37_PO, oDrive_Param := "Station_MOVIKIT".MSt37_PI)
   END_RUNG
   // the same network as SCL:
   "Drivers_To_Move_Pallet"(HW_Driver := "MST37~Module_I_O_(05_words)_1",
                           Reset := "HMI_Pallets".Reset_Drivers,
                           iDrive_Param := "Station_MOVIKIT".MSt37_PO,
                           oDrive_Param := "Station_MOVIKIT".MSt37_PI);
END_REGION

REGION Network 49: MST38
   RUNG wire#powerrail
      "Drivers_To_Move_Pallet"(HW_Driver := "MST38~Module_I_O_(05_words)_1", Reset := "HMI_Pallets".Reset_Drivers, iDrive_Param := "Station_MOVIKIT".MSt38_PO, oDrive_Param := "Station_MOVIKIT".MSt38_PI)
   END_RUNG
   // the same network as SCL:
   "Drivers_To_Move_Pallet"(HW_Driver := "MST38~Module_I_O_(05_words)_1",
                           Reset := "HMI_Pallets".Reset_Drivers,
                           iDrive_Param := "Station_MOVIKIT".MSt38_PO,
                           oDrive_Param := "Station_MOVIKIT".MSt38_PI);
END_REGION

REGION Network 50 (SCL): Clean Movment
   "Clean_Movment"(Arr := "HMI_Pallets".Run_Command_left_ROW1);
   "Clean_Movment"(Arr := "HMI_Pallets".Run_Command_left_ROW2);
   "Clean_Movment"(Arr := "HMI_Pallets".Run_Command_left_ROW3);
   "Clean_Movment"(Arr := "HMI_Pallets".Run_Command_left_ROW4);

   "Clean_Movment"(Arr := "HMI_Pallets".Run_Command_right_ROW1);
   "Clean_Movment"(Arr := "HMI_Pallets".Run_Command_right_ROW2);
   "Clean_Movment"(Arr := "HMI_Pallets".Run_Command_right_ROW3);
   "Clean_Movment"(Arr := "HMI_Pallets".Run_Command_right_ROW4);
END_REGION

REGION Network 51: ST13->ST14
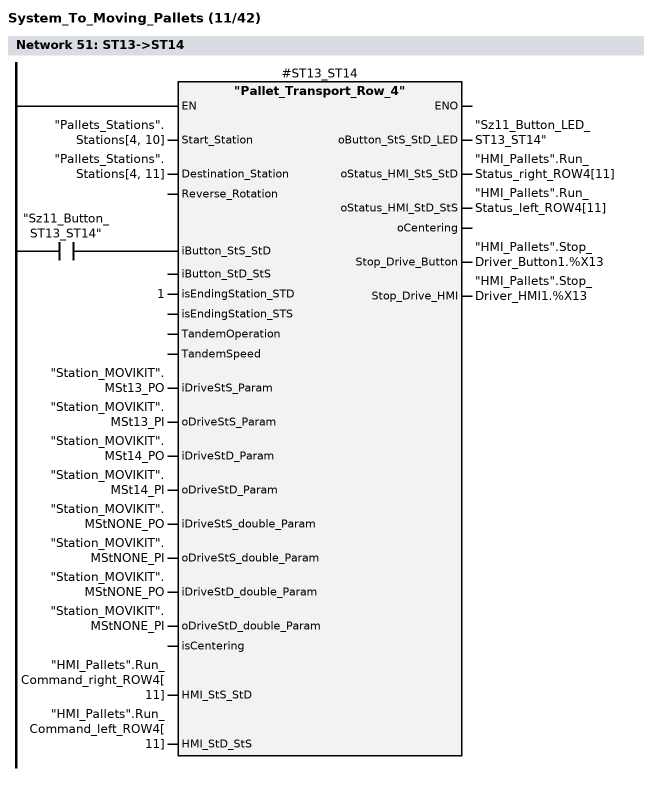
   RUNG wire#powerrail
      #ST13_ST14(iButton_StS_StD := wire#w1, Start_Station := "Pallets_Stations".Stations[4, 10], Destination_Station := "Pallets_Stations".Stations[4, 11], Reverse_Rotation :=, iButton_StD_StS :=, isEndingStation_STD := 1, isEndingStation_STS :=, TandemOperation :=, TandemSpeed :=, iDriveStS_Param := "Station_MOVIKIT".MSt13_PO, oDriveStS_Param := "Station_MOVIKIT".MSt13_PI, iDriveStD_Param := "Station_MOVIKIT".MSt14_PO, oDriveStD_Param := "Station_MOVIKIT".MSt14_PI, iDriveStS_double_Param := "Station_MOVIKIT".MStNONE_PO, oDriveStS_double_Param := "Station_MOVIKIT".MStNONE_PI, iDriveStD_double_Param := "Station_MOVIKIT".MStNONE_PO, oDriveStD_double_Param := "Station_MOVIKIT".MStNONE_PI, isCentering :=, HMI_StS_StD := "HMI_Pallets".Run_Command_right_ROW4[11], HMI_StD_StS := "HMI_Pallets".Run_Command_left_ROW4[11], oButton_StS_StD_LED => "Sz11_Button_LED_ST13_ST14", oStatus_HMI_StS_StD => "HMI_Pallets".Run_Status_right_ROW4[11], oStatus_HMI_StD_StS => "HMI_Pallets".Run_Status_left_ROW4[11], oCentering =>, Stop_Drive_Button => "HMI_Pallets".Stop_Driver_Button1.%X13, Stop_Drive_HMI => "HMI_Pallets".Stop_Driver_HMI1.%X13)
   END_RUNG
   RUNG wire#powerrail
      Contact( "Sz11_Button_ST13_ST14" )
   END_RUNG wire#w1
   // the same network as SCL:
   #ST13_ST14(Start_Station := "Pallets_Stations".Stations[4, 10],   // "Pallet_Transport_Row_4"
              Destination_Station := "Pallets_Stations".Stations[4, 11],
              iButton_StS_StD := "Sz11_Button_ST13_ST14",
              isEndingStation_STD := 1,
              iDriveStS_Param := "Station_MOVIKIT".MSt13_PO,
              oDriveStS_Param := "Station_MOVIKIT".MSt13_PI,
              iDriveStD_Param := "Station_MOVIKIT".MSt14_PO,
              oDriveStD_Param := "Station_MOVIKIT".MSt14_PI,
              iDriveStS_double_Param := "Station_MOVIKIT".MStNONE_PO,
              oDriveStS_double_Param := "Station_MOVIKIT".MStNONE_PI,
              iDriveStD_double_Param := "Station_MOVIKIT".MStNONE_PO,
              oDriveStD_double_Param := "Station_MOVIKIT".MStNONE_PI,
              HMI_StS_StD := "HMI_Pallets".Run_Command_right_ROW4[11],
              HMI_StD_StS := "HMI_Pallets".Run_Command_left_ROW4[11],
              oButton_StS_StD_LED => "Sz11_Button_LED_ST13_ST14",
              oStatus_HMI_StS_StD => "HMI_Pallets".Run_Status_right_ROW4[11],
              oStatus_HMI_StD_StS => "HMI_Pallets".Run_Status_left_ROW4[11],
              Stop_Drive_Button => "HMI_Pallets".Stop_Driver_Button1.%X13,
              Stop_Drive_HMI => "HMI_Pallets".Stop_Driver_HMI1.%X13);
END_REGION

REGION Network 52: ST12->ST13
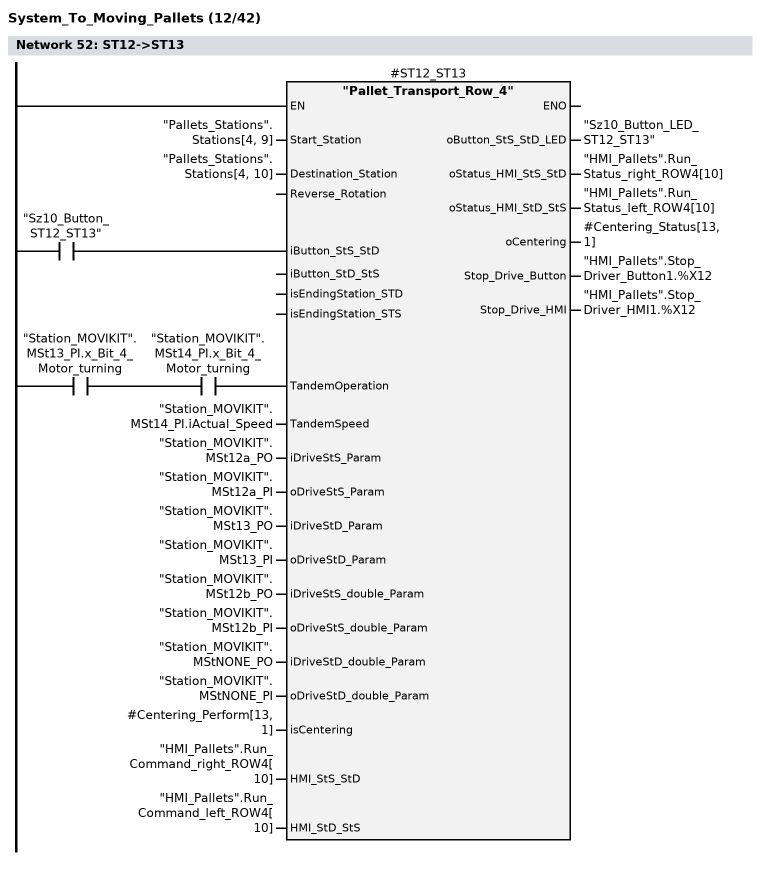
   RUNG wire#powerrail
      #ST12_ST13(iButton_StS_StD := wire#w1, TandemOperation := wire#w2, Start_Station := "Pallets_Stations".Stations[4, 9], Destination_Station := "Pallets_Stations".Stations[4, 10], Reverse_Rotation :=, iButton_StD_StS :=, isEndingStation_STD :=, isEndingStation_STS :=, TandemSpeed := "Station_MOVIKIT".MSt14_PI.iActual_Speed, iDriveStS_Param := "Station_MOVIKIT".MSt12a_PO, oDriveStS_Param := "Station_MOVIKIT".MSt12a_PI, iDriveStD_Param := "Station_MOVIKIT".MSt13_PO, oDriveStD_Param := "Station_MOVIKIT".MSt13_PI, iDriveStS_double_Param := "Station_MOVIKIT".MSt12b_PO, oDriveStS_double_Param := "Station_MOVIKIT".MSt12b_PI, iDriveStD_double_Param := "Station_MOVIKIT".MStNONE_PO, oDriveStD_double_Param := "Station_MOVIKIT".MStNONE_PI, isCentering := #Centering_Perform[13, 1], HMI_StS_StD := "HMI_Pallets".Run_Command_right_ROW4[10], HMI_StD_StS := "HMI_Pallets".Run_Command_left_ROW4[10], oButton_StS_StD_LED => "Sz10_Button_LED_ST12_ST13", oStatus_HMI_StS_StD => "HMI_Pallets".Run_Status_right_ROW4[10], oStatus_HMI_StD_StS => "HMI_Pallets".Run_Status_left_ROW4[10], oCentering => #Centering_Status[13, 1], Stop_Drive_Button => "HMI_Pallets".Stop_Driver_Button1.%X12, Stop_Drive_HMI => "HMI_Pallets".Stop_Driver_HMI1.%X12)
   END_RUNG
   RUNG wire#powerrail
      Contact( "Sz10_Button_ST12_ST13" )
   END_RUNG wire#w1
   RUNG wire#powerrail
      Contact( "Station_MOVIKIT".MSt13_PI.x_Bit_4_Motor_turning )
      Contact( "Station_MOVIKIT".MSt14_PI.x_Bit_4_Motor_turning )
   END_RUNG wire#w2
   // the same network as SCL:
   #ST12_ST13(Start_Station := "Pallets_Stations".Stations[4, 9],   // "Pallet_Transport_Row_4"
              Destination_Station := "Pallets_Stations".Stations[4, 10],
              iButton_StS_StD := "Sz10_Button_ST12_ST13",
              TandemOperation := "Station_MOVIKIT".MSt13_PI.x_Bit_4_Motor_turning AND "Station_MOVIKIT".MSt14_PI.x_Bit_4_Motor_turning,
              TandemSpeed := "Station_MOVIKIT".MSt14_PI.iActual_Speed,
              iDriveStS_Param := "Station_MOVIKIT".MSt12a_PO,
              oDriveStS_Param := "Station_MOVIKIT".MSt12a_PI,
              iDriveStD_Param := "Station_MOVIKIT".MSt13_PO,
              oDriveStD_Param := "Station_MOVIKIT".MSt13_PI,
              iDriveStS_double_Param := "Station_MOVIKIT".MSt12b_PO,
              oDriveStS_double_Param := "Station_MOVIKIT".MSt12b_PI,
              iDriveStD_double_Param := "Station_MOVIKIT".MStNONE_PO,
              oDriveStD_double_Param := "Station_MOVIKIT".MStNONE_PI,
              isCentering := #Centering_Perform[13, 1],
              HMI_StS_StD := "HMI_Pallets".Run_Command_right_ROW4[10],
              HMI_StD_StS := "HMI_Pallets".Run_Command_left_ROW4[10],
              oButton_StS_StD_LED => "Sz10_Button_LED_ST12_ST13",
              oStatus_HMI_StS_StD => "HMI_Pallets".Run_Status_right_ROW4[10],
              oStatus_HMI_StD_StS => "HMI_Pallets".Run_Status_left_ROW4[10],
              oCentering => #Centering_Status[13, 1],
              Stop_Drive_Button => "HMI_Pallets".Stop_Driver_Button1.%X12,
              Stop_Drive_HMI => "HMI_Pallets".Stop_Driver_HMI1.%X12);
END_REGION

REGION Network 53: ST11->ST12
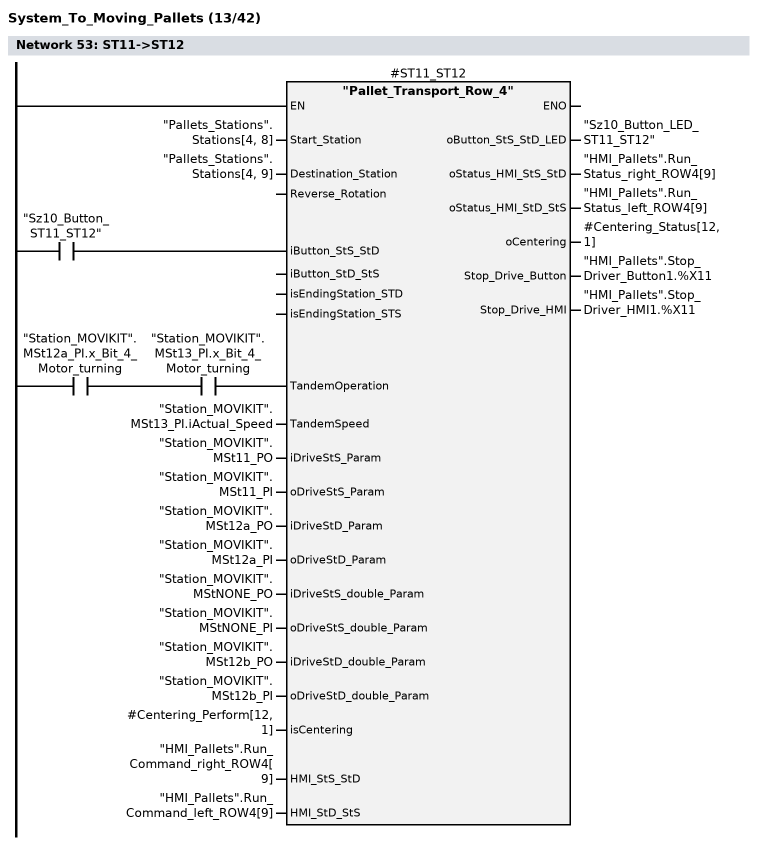
   RUNG wire#powerrail
      #ST11_ST12(iButton_StS_StD := wire#w1, TandemOperation := wire#w2, Start_Station := "Pallets_Stations".Stations[4, 8], Destination_Station := "Pallets_Stations".Stations[4, 9], Reverse_Rotation :=, iButton_StD_StS :=, isEndingStation_STD :=, isEndingStation_STS :=, TandemSpeed := "Station_MOVIKIT".MSt13_PI.iActual_Speed, iDriveStS_Param := "Station_MOVIKIT".MSt11_PO, oDriveStS_Param := "Station_MOVIKIT".MSt11_PI, iDriveStD_Param := "Station_MOVIKIT".MSt12a_PO, oDriveStD_Param := "Station_MOVIKIT".MSt12a_PI, iDriveStS_double_Param := "Station_MOVIKIT".MStNONE_PO, oDriveStS_double_Param := "Station_MOVIKIT".MStNONE_PI, iDriveStD_double_Param := "Station_MOVIKIT".MSt12b_PO, oDriveStD_double_Param := "Station_MOVIKIT".MSt12b_PI, isCentering := #Centering_Perform[12, 1], HMI_StS_StD := "HMI_Pallets".Run_Command_right_ROW4[9], HMI_StD_StS := "HMI_Pallets".Run_Command_left_ROW4[9], oButton_StS_StD_LED => "Sz10_Button_LED_ST11_ST12", oStatus_HMI_StS_StD => "HMI_Pallets".Run_Status_right_ROW4[9], oStatus_HMI_StD_StS => "HMI_Pallets".Run_Status_left_ROW4[9], oCentering => #Centering_Status[12, 1], Stop_Drive_Button => "HMI_Pallets".Stop_Driver_Button1.%X11, Stop_Drive_HMI => "HMI_Pallets".Stop_Driver_HMI1.%X11)
   END_RUNG
   RUNG wire#powerrail
      Contact( "Sz10_Button_ST11_ST12" )
   END_RUNG wire#w1
   RUNG wire#powerrail
      Contact( "Station_MOVIKIT".MSt12a_PI.x_Bit_4_Motor_turning )
      Contact( "Station_MOVIKIT".MSt13_PI.x_Bit_4_Motor_turning )
   END_RUNG wire#w2
   // the same network as SCL:
   #ST11_ST12(Start_Station := "Pallets_Stations".Stations[4, 8],   // "Pallet_Transport_Row_4"
              Destination_Station := "Pallets_Stations".Stations[4, 9],
              iButton_StS_StD := "Sz10_Button_ST11_ST12",
              TandemOperation := "Station_MOVIKIT".MSt12a_PI.x_Bit_4_Motor_turning AND "Station_MOVIKIT".MSt13_PI.x_Bit_4_Motor_turning,
              TandemSpeed := "Station_MOVIKIT".MSt13_PI.iActual_Speed,
              iDriveStS_Param := "Station_MOVIKIT".MSt11_PO,
              oDriveStS_Param := "Station_MOVIKIT".MSt11_PI,
              iDriveStD_Param := "Station_MOVIKIT".MSt12a_PO,
              oDriveStD_Param := "Station_MOVIKIT".MSt12a_PI,
              iDriveStS_double_Param := "Station_MOVIKIT".MStNONE_PO,
              oDriveStS_double_Param := "Station_MOVIKIT".MStNONE_PI,
              iDriveStD_double_Param := "Station_MOVIKIT".MSt12b_PO,
              oDriveStD_double_Param := "Station_MOVIKIT".MSt12b_PI,
              isCentering := #Centering_Perform[12, 1],
              HMI_StS_StD := "HMI_Pallets".Run_Command_right_ROW4[9],
              HMI_StD_StS := "HMI_Pallets".Run_Command_left_ROW4[9],
              oButton_StS_StD_LED => "Sz10_Button_LED_ST11_ST12",
              oStatus_HMI_StS_StD => "HMI_Pallets".Run_Status_right_ROW4[9],
              oStatus_HMI_StD_StS => "HMI_Pallets".Run_Status_left_ROW4[9],
              oCentering => #Centering_Status[12, 1],
              Stop_Drive_Button => "HMI_Pallets".Stop_Driver_Button1.%X11,
              Stop_Drive_HMI => "HMI_Pallets".Stop_Driver_HMI1.%X11);
END_REGION

REGION Network 54: ST10->ST11
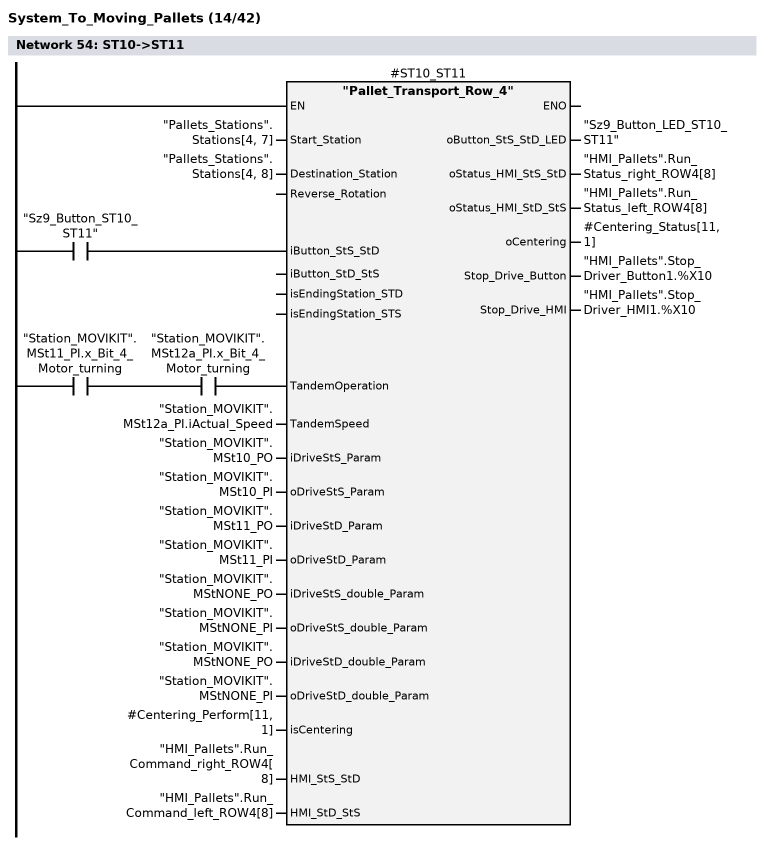
   RUNG wire#powerrail
      #ST10_ST11(iButton_StS_StD := wire#w1, TandemOperation := wire#w2, Start_Station := "Pallets_Stations".Stations[4, 7], Destination_Station := "Pallets_Stations".Stations[4, 8], Reverse_Rotation :=, iButton_StD_StS :=, isEndingStation_STD :=, isEndingStation_STS :=, TandemSpeed := "Station_MOVIKIT".MSt12a_PI.iActual_Speed, iDriveStS_Param := "Station_MOVIKIT".MSt10_PO, oDriveStS_Param := "Station_MOVIKIT".MSt10_PI, iDriveStD_Param := "Station_MOVIKIT".MSt11_PO, oDriveStD_Param := "Station_MOVIKIT".MSt11_PI, iDriveStS_double_Param := "Station_MOVIKIT".MStNONE_PO, oDriveStS_double_Param := "Station_MOVIKIT".MStNONE_PI, iDriveStD_double_Param := "Station_MOVIKIT".MStNONE_PO, oDriveStD_double_Param := "Station_MOVIKIT".MStNONE_PI, isCentering := #Centering_Perform[11, 1], HMI_StS_StD := "HMI_Pallets".Run_Command_right_ROW4[8], HMI_StD_StS := "HMI_Pallets".Run_Command_left_ROW4[8], oButton_StS_StD_LED => "Sz9_Button_LED_ST10_ST11", oStatus_HMI_StS_StD => "HMI_Pallets".Run_Status_right_ROW4[8], oStatus_HMI_StD_StS => "HMI_Pallets".Run_Status_left_ROW4[8], oCentering => #Centering_Status[11, 1], Stop_Drive_Button => "HMI_Pallets".Stop_Driver_Button1.%X10, Stop_Drive_HMI => "HMI_Pallets".Stop_Driver_HMI1.%X10)
   END_RUNG
   RUNG wire#powerrail
      Contact( "Sz9_Button_ST10_ST11" )
   END_RUNG wire#w1
   RUNG wire#powerrail
      Contact( "Station_MOVIKIT".MSt11_PI.x_Bit_4_Motor_turning )
      Contact( "Station_MOVIKIT".MSt12a_PI.x_Bit_4_Motor_turning )
   END_RUNG wire#w2
   // the same network as SCL:
   #ST10_ST11(Start_Station := "Pallets_Stations".Stations[4, 7],   // "Pallet_Transport_Row_4"
              Destination_Station := "Pallets_Stations".Stations[4, 8],
              iButton_StS_StD := "Sz9_Button_ST10_ST11",
              TandemOperation := "Station_MOVIKIT".MSt11_PI.x_Bit_4_Motor_turning AND "Station_MOVIKIT".MSt12a_PI.x_Bit_4_Motor_turning,
              TandemSpeed := "Station_MOVIKIT".MSt12a_PI.iActual_Speed,
              iDriveStS_Param := "Station_MOVIKIT".MSt10_PO,
              oDriveStS_Param := "Station_MOVIKIT".MSt10_PI,
              iDriveStD_Param := "Station_MOVIKIT".MSt11_PO,
              oDriveStD_Param := "Station_MOVIKIT".MSt11_PI,
              iDriveStS_double_Param := "Station_MOVIKIT".MStNONE_PO,
              oDriveStS_double_Param := "Station_MOVIKIT".MStNONE_PI,
              iDriveStD_double_Param := "Station_MOVIKIT".MStNONE_PO,
              oDriveStD_double_Param := "Station_MOVIKIT".MStNONE_PI,
              isCentering := #Centering_Perform[11, 1],
              HMI_StS_StD := "HMI_Pallets".Run_Command_right_ROW4[8],
              HMI_StD_StS := "HMI_Pallets".Run_Command_left_ROW4[8],
              oButton_StS_StD_LED => "Sz9_Button_LED_ST10_ST11",
              oStatus_HMI_StS_StD => "HMI_Pallets".Run_Status_right_ROW4[8],
              oStatus_HMI_StD_StS => "HMI_Pallets".Run_Status_left_ROW4[8],
              oCentering => #Centering_Status[11, 1],
              Stop_Drive_Button => "HMI_Pallets".Stop_Driver_Button1.%X10,
              Stop_Drive_HMI => "HMI_Pallets".Stop_Driver_HMI1.%X10);
END_REGION

REGION Network 55: ST09->ST10
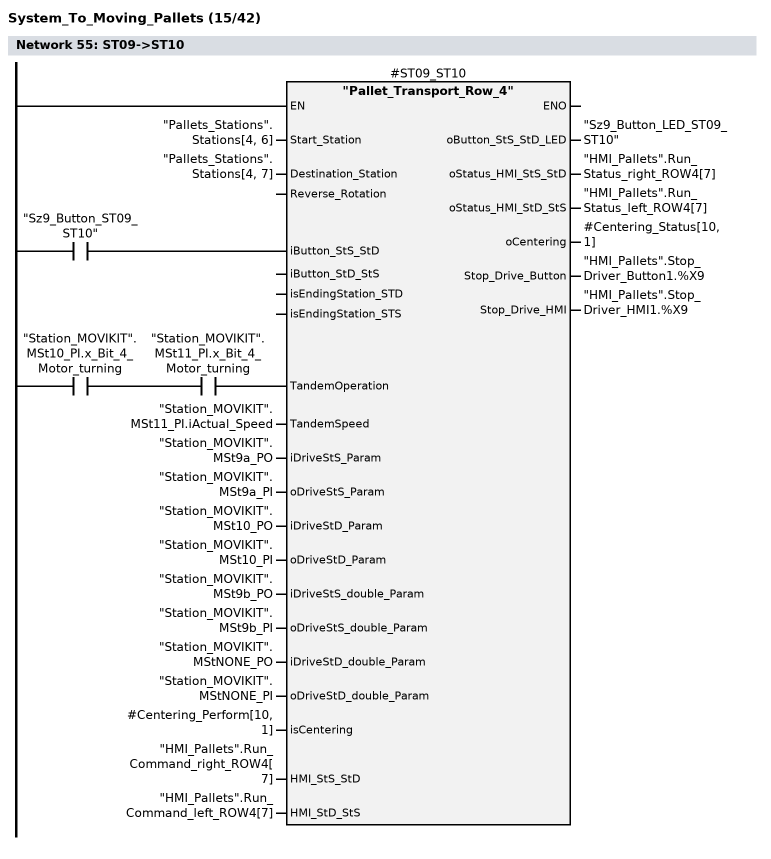
   RUNG wire#powerrail
      #ST09_ST10(iButton_StS_StD := wire#w1, TandemOperation := wire#w2, Start_Station := "Pallets_Stations".Stations[4, 6], Destination_Station := "Pallets_Stations".Stations[4, 7], Reverse_Rotation :=, iButton_StD_StS :=, isEndingStation_STD :=, isEndingStation_STS :=, TandemSpeed := "Station_MOVIKIT".MSt11_PI.iActual_Speed, iDriveStS_Param := "Station_MOVIKIT".MSt9a_PO, oDriveStS_Param := "Station_MOVIKIT".MSt9a_PI, iDriveStD_Param := "Station_MOVIKIT".MSt10_PO, oDriveStD_Param := "Station_MOVIKIT".MSt10_PI, iDriveStS_double_Param := "Station_MOVIKIT".MSt9b_PO, oDriveStS_double_Param := "Station_MOVIKIT".MSt9b_PI, iDriveStD_double_Param := "Station_MOVIKIT".MStNONE_PO, oDriveStD_double_Param := "Station_MOVIKIT".MStNONE_PI, isCentering := #Centering_Perform[10, 1], HMI_StS_StD := "HMI_Pallets".Run_Command_right_ROW4[7], HMI_StD_StS := "HMI_Pallets".Run_Command_left_ROW4[7], oButton_StS_StD_LED => "Sz9_Button_LED_ST09_ST10", oStatus_HMI_StS_StD => "HMI_Pallets".Run_Status_right_ROW4[7], oStatus_HMI_StD_StS => "HMI_Pallets".Run_Status_left_ROW4[7], oCentering => #Centering_Status[10, 1], Stop_Drive_Button => "HMI_Pallets".Stop_Driver_Button1.%X9, Stop_Drive_HMI => "HMI_Pallets".Stop_Driver_HMI1.%X9)
   END_RUNG
   RUNG wire#powerrail
      Contact( "Sz9_Button_ST09_ST10" )
   END_RUNG wire#w1
   RUNG wire#powerrail
      Contact( "Station_MOVIKIT".MSt10_PI.x_Bit_4_Motor_turning )
      Contact( "Station_MOVIKIT".MSt11_PI.x_Bit_4_Motor_turning )
   END_RUNG wire#w2
   // the same network as SCL:
   #ST09_ST10(Start_Station := "Pallets_Stations".Stations[4, 6],   // "Pallet_Transport_Row_4"
              Destination_Station := "Pallets_Stations".Stations[4, 7],
              iButton_StS_StD := "Sz9_Button_ST09_ST10",
              TandemOperation := "Station_MOVIKIT".MSt10_PI.x_Bit_4_Motor_turning AND "Station_MOVIKIT".MSt11_PI.x_Bit_4_Motor_turning,
              TandemSpeed := "Station_MOVIKIT".MSt11_PI.iActual_Speed,
              iDriveStS_Param := "Station_MOVIKIT".MSt9a_PO,
              oDriveStS_Param := "Station_MOVIKIT".MSt9a_PI,
              iDriveStD_Param := "Station_MOVIKIT".MSt10_PO,
              oDriveStD_Param := "Station_MOVIKIT".MSt10_PI,
              iDriveStS_double_Param := "Station_MOVIKIT".MSt9b_PO,
              oDriveStS_double_Param := "Station_MOVIKIT".MSt9b_PI,
              iDriveStD_double_Param := "Station_MOVIKIT".MStNONE_PO,
              oDriveStD_double_Param := "Station_MOVIKIT".MStNONE_PI,
              isCentering := #Centering_Perform[10, 1],
              HMI_StS_StD := "HMI_Pallets".Run_Command_right_ROW4[7],
              HMI_StD_StS := "HMI_Pallets".Run_Command_left_ROW4[7],
              oButton_StS_StD_LED => "Sz9_Button_LED_ST09_ST10",
              oStatus_HMI_StS_StD => "HMI_Pallets".Run_Status_right_ROW4[7],
              oStatus_HMI_StD_StS => "HMI_Pallets".Run_Status_left_ROW4[7],
              oCentering => #Centering_Status[10, 1],
              Stop_Drive_Button => "HMI_Pallets".Stop_Driver_Button1.%X9,
              Stop_Drive_HMI => "HMI_Pallets".Stop_Driver_HMI1.%X9);
END_REGION

REGION Network 56: ST08->ST09
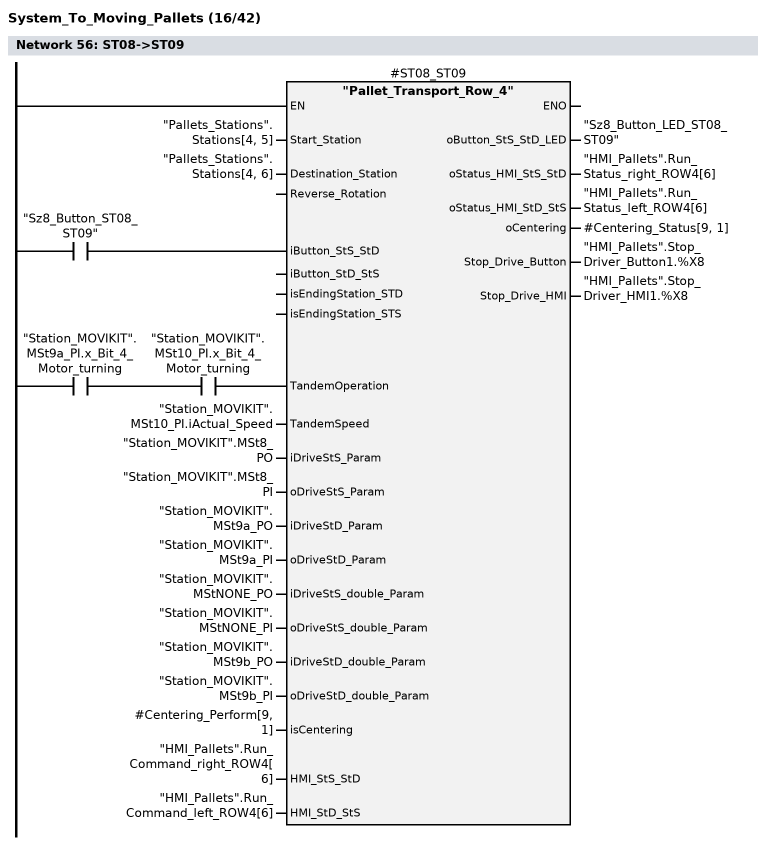
   RUNG wire#powerrail
      #ST08_ST09(iButton_StS_StD := wire#w1, TandemOperation := wire#w2, Start_Station := "Pallets_Stations".Stations[4, 5], Destination_Station := "Pallets_Stations".Stations[4, 6], Reverse_Rotation :=, iButton_StD_StS :=, isEndingStation_STD :=, isEndingStation_STS :=, TandemSpeed := "Station_MOVIKIT".MSt10_PI.iActual_Speed, iDriveStS_Param := "Station_MOVIKIT".MSt8_PO, oDriveStS_Param := "Station_MOVIKIT".MSt8_PI, iDriveStD_Param := "Station_MOVIKIT".MSt9a_PO, oDriveStD_Param := "Station_MOVIKIT".MSt9a_PI, iDriveStS_double_Param := "Station_MOVIKIT".MStNONE_PO, oDriveStS_double_Param := "Station_MOVIKIT".MStNONE_PI, iDriveStD_double_Param := "Station_MOVIKIT".MSt9b_PO, oDriveStD_double_Param := "Station_MOVIKIT".MSt9b_PI, isCentering := #Centering_Perform[9, 1], HMI_StS_StD := "HMI_Pallets".Run_Command_right_ROW4[6], HMI_StD_StS := "HMI_Pallets".Run_Command_left_ROW4[6], oButton_StS_StD_LED => "Sz8_Button_LED_ST08_ST09", oStatus_HMI_StS_StD => "HMI_Pallets".Run_Status_right_ROW4[6], oStatus_HMI_StD_StS => "HMI_Pallets".Run_Status_left_ROW4[6], oCentering => #Centering_Status[9, 1], Stop_Drive_Button => "HMI_Pallets".Stop_Driver_Button1.%X8, Stop_Drive_HMI => "HMI_Pallets".Stop_Driver_HMI1.%X8)
   END_RUNG
   RUNG wire#powerrail
      Contact( "Sz8_Button_ST08_ST09" )
   END_RUNG wire#w1
   RUNG wire#powerrail
      Contact( "Station_MOVIKIT".MSt9a_PI.x_Bit_4_Motor_turning )
      Contact( "Station_MOVIKIT".MSt10_PI.x_Bit_4_Motor_turning )
   END_RUNG wire#w2
   // the same network as SCL:
   #ST08_ST09(Start_Station := "Pallets_Stations".Stations[4, 5],   // "Pallet_Transport_Row_4"
              Destination_Station := "Pallets_Stations".Stations[4, 6],
              iButton_StS_StD := "Sz8_Button_ST08_ST09",
              TandemOperation := "Station_MOVIKIT".MSt9a_PI.x_Bit_4_Motor_turning AND "Station_MOVIKIT".MSt10_PI.x_Bit_4_Motor_turning,
              TandemSpeed := "Station_MOVIKIT".MSt10_PI.iActual_Speed,
              iDriveStS_Param := "Station_MOVIKIT".MSt8_PO,
              oDriveStS_Param := "Station_MOVIKIT".MSt8_PI,
              iDriveStD_Param := "Station_MOVIKIT".MSt9a_PO,
              oDriveStD_Param := "Station_MOVIKIT".MSt9a_PI,
              iDriveStS_double_Param := "Station_MOVIKIT".MStNONE_PO,
              oDriveStS_double_Param := "Station_MOVIKIT".MStNONE_PI,
              iDriveStD_double_Param := "Station_MOVIKIT".MSt9b_PO,
              oDriveStD_double_Param := "Station_MOVIKIT".MSt9b_PI,
              isCentering := #Centering_Perform[9, 1],
              HMI_StS_StD := "HMI_Pallets".Run_Command_right_ROW4[6],
              HMI_StD_StS := "HMI_Pallets".Run_Command_left_ROW4[6],
              oButton_StS_StD_LED => "Sz8_Button_LED_ST08_ST09",
              oStatus_HMI_StS_StD => "HMI_Pallets".Run_Status_right_ROW4[6],
              oStatus_HMI_StD_StS => "HMI_Pallets".Run_Status_left_ROW4[6],
              oCentering => #Centering_Status[9, 1],
              Stop_Drive_Button => "HMI_Pallets".Stop_Driver_Button1.%X8,
              Stop_Drive_HMI => "HMI_Pallets".Stop_Driver_HMI1.%X8);
END_REGION

REGION Network 57: ST07->ST08
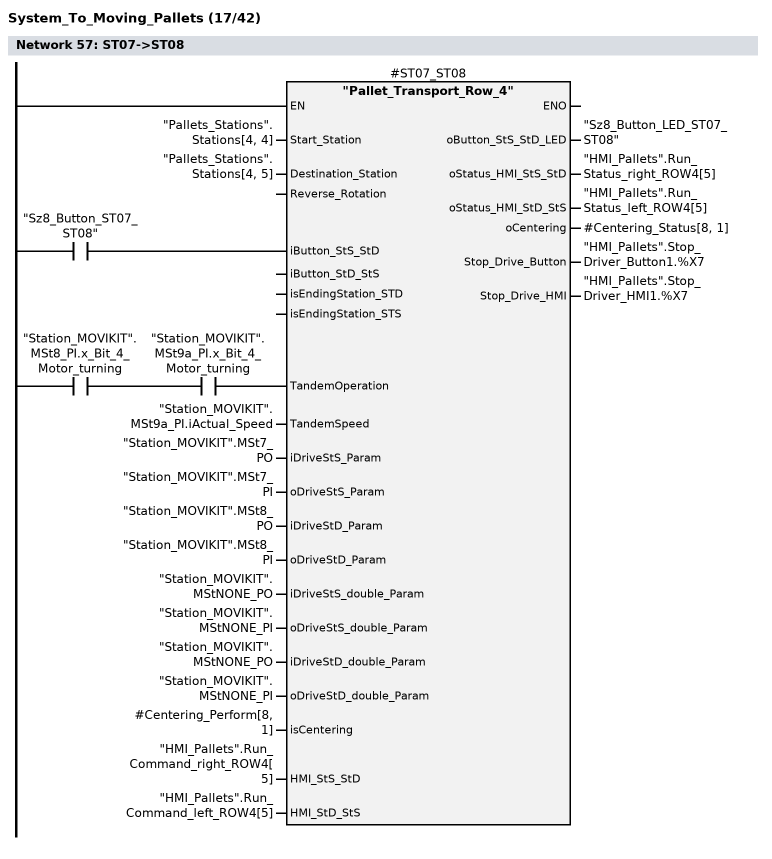
   RUNG wire#powerrail
      #ST07_ST08(iButton_StS_StD := wire#w1, TandemOperation := wire#w2, Start_Station := "Pallets_Stations".Stations[4, 4], Destination_Station := "Pallets_Stations".Stations[4, 5], Reverse_Rotation :=, iButton_StD_StS :=, isEndingStation_STD :=, isEndingStation_STS :=, TandemSpeed := "Station_MOVIKIT".MSt9a_PI.iActual_Speed, iDriveStS_Param := "Station_MOVIKIT".MSt7_PO, oDriveStS_Param := "Station_MOVIKIT".MSt7_PI, iDriveStD_Param := "Station_MOVIKIT".MSt8_PO, oDriveStD_Param := "Station_MOVIKIT".MSt8_PI, iDriveStS_double_Param := "Station_MOVIKIT".MStNONE_PO, oDriveStS_double_Param := "Station_MOVIKIT".MStNONE_PI, iDriveStD_double_Param := "Station_MOVIKIT".MStNONE_PO, oDriveStD_double_Param := "Station_MOVIKIT".MStNONE_PI, isCentering := #Centering_Perform[8, 1], HMI_StS_StD := "HMI_Pallets".Run_Command_right_ROW4[5], HMI_StD_StS := "HMI_Pallets".Run_Command_left_ROW4[5], oButton_StS_StD_LED => "Sz8_Button_LED_ST07_ST08", oStatus_HMI_StS_StD => "HMI_Pallets".Run_Status_right_ROW4[5], oStatus_HMI_StD_StS => "HMI_Pallets".Run_Status_left_ROW4[5], oCentering => #Centering_Status[8, 1], Stop_Drive_Button => "HMI_Pallets".Stop_Driver_Button1.%X7, Stop_Drive_HMI => "HMI_Pallets".Stop_Driver_HMI1.%X7)
   END_RUNG
   RUNG wire#powerrail
      Contact( "Sz8_Button_ST07_ST08" )
   END_RUNG wire#w1
   RUNG wire#powerrail
      Contact( "Station_MOVIKIT".MSt8_PI.x_Bit_4_Motor_turning )
      Contact( "Station_MOVIKIT".MSt9a_PI.x_Bit_4_Motor_turning )
   END_RUNG wire#w2
   // the same network as SCL:
   #ST07_ST08(Start_Station := "Pallets_Stations".Stations[4, 4],   // "Pallet_Transport_Row_4"
              Destination_Station := "Pallets_Stations".Stations[4, 5],
              iButton_StS_StD := "Sz8_Button_ST07_ST08",
              TandemOperation := "Station_MOVIKIT".MSt8_PI.x_Bit_4_Motor_turning AND "Station_MOVIKIT".MSt9a_PI.x_Bit_4_Motor_turning,
              TandemSpeed := "Station_MOVIKIT".MSt9a_PI.iActual_Speed,
              iDriveStS_Param := "Station_MOVIKIT".MSt7_PO,
              oDriveStS_Param := "Station_MOVIKIT".MSt7_PI,
              iDriveStD_Param := "Station_MOVIKIT".MSt8_PO,
              oDriveStD_Param := "Station_MOVIKIT".MSt8_PI,
              iDriveStS_double_Param := "Station_MOVIKIT".MStNONE_PO,
              oDriveStS_double_Param := "Station_MOVIKIT".MStNONE_PI,
              iDriveStD_double_Param := "Station_MOVIKIT".MStNONE_PO,
              oDriveStD_double_Param := "Station_MOVIKIT".MStNONE_PI,
              isCentering := #Centering_Perform[8, 1],
              HMI_StS_StD := "HMI_Pallets".Run_Command_right_ROW4[5],
              HMI_StD_StS := "HMI_Pallets".Run_Command_left_ROW4[5],
              oButton_StS_StD_LED => "Sz8_Button_LED_ST07_ST08",
              oStatus_HMI_StS_StD => "HMI_Pallets".Run_Status_right_ROW4[5],
              oStatus_HMI_StD_StS => "HMI_Pallets".Run_Status_left_ROW4[5],
              oCentering => #Centering_Status[8, 1],
              Stop_Drive_Button => "HMI_Pallets".Stop_Driver_Button1.%X7,
              Stop_Drive_HMI => "HMI_Pallets".Stop_Driver_HMI1.%X7);
END_REGION

REGION Network 58: ST06->ST07
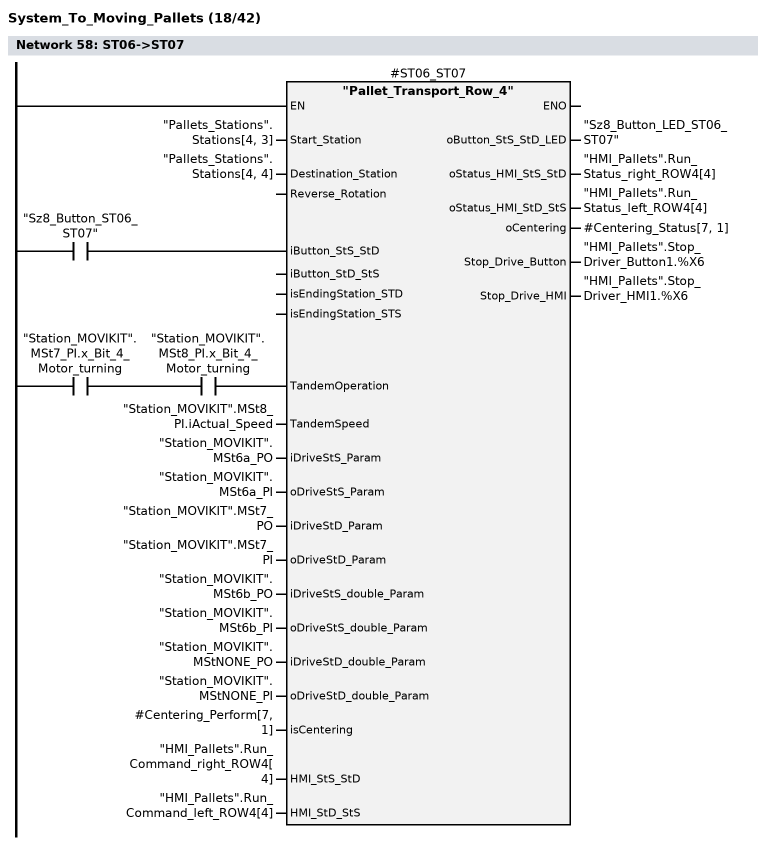
   RUNG wire#powerrail
      #ST06_ST07(iButton_StS_StD := wire#w1, TandemOperation := wire#w2, Start_Station := "Pallets_Stations".Stations[4, 3], Destination_Station := "Pallets_Stations".Stations[4, 4], Reverse_Rotation :=, iButton_StD_StS :=, isEndingStation_STD :=, isEndingStation_STS :=, TandemSpeed := "Station_MOVIKIT".MSt8_PI.iActual_Speed, iDriveStS_Param := "Station_MOVIKIT".MSt6a_PO, oDriveStS_Param := "Station_MOVIKIT".MSt6a_PI, iDriveStD_Param := "Station_MOVIKIT".MSt7_PO, oDriveStD_Param := "Station_MOVIKIT".MSt7_PI, iDriveStS_double_Param := "Station_MOVIKIT".MSt6b_PO, oDriveStS_double_Param := "Station_MOVIKIT".MSt6b_PI, iDriveStD_double_Param := "Station_MOVIKIT".MStNONE_PO, oDriveStD_double_Param := "Station_MOVIKIT".MStNONE_PI, isCentering := #Centering_Perform[7, 1], HMI_StS_StD := "HMI_Pallets".Run_Command_right_ROW4[4], HMI_StD_StS := "HMI_Pallets".Run_Command_left_ROW4[4], oButton_StS_StD_LED => "Sz8_Button_LED_ST06_ST07", oStatus_HMI_StS_StD => "HMI_Pallets".Run_Status_right_ROW4[4], oStatus_HMI_StD_StS => "HMI_Pallets".Run_Status_left_ROW4[4], oCentering => #Centering_Status[7, 1], Stop_Drive_Button => "HMI_Pallets".Stop_Driver_Button1.%X6, Stop_Drive_HMI => "HMI_Pallets".Stop_Driver_HMI1.%X6)
   END_RUNG
   RUNG wire#powerrail
      Contact( "Sz8_Button_ST06_ST07" )
   END_RUNG wire#w1
   RUNG wire#powerrail
      Contact( "Station_MOVIKIT".MSt7_PI.x_Bit_4_Motor_turning )
      Contact( "Station_MOVIKIT".MSt8_PI.x_Bit_4_Motor_turning )
   END_RUNG wire#w2
   // the same network as SCL:
   #ST06_ST07(Start_Station := "Pallets_Stations".Stations[4, 3],   // "Pallet_Transport_Row_4"
              Destination_Station := "Pallets_Stations".Stations[4, 4],
              iButton_StS_StD := "Sz8_Button_ST06_ST07",
              TandemOperation := "Station_MOVIKIT".MSt7_PI.x_Bit_4_Motor_turning AND "Station_MOVIKIT".MSt8_PI.x_Bit_4_Motor_turning,
              TandemSpeed := "Station_MOVIKIT".MSt8_PI.iActual_Speed,
              iDriveStS_Param := "Station_MOVIKIT".MSt6a_PO,
              oDriveStS_Param := "Station_MOVIKIT".MSt6a_PI,
              iDriveStD_Param := "Station_MOVIKIT".MSt7_PO,
              oDriveStD_Param := "Station_MOVIKIT".MSt7_PI,
              iDriveStS_double_Param := "Station_MOVIKIT".MSt6b_PO,
              oDriveStS_double_Param := "Station_MOVIKIT".MSt6b_PI,
              iDriveStD_double_Param := "Station_MOVIKIT".MStNONE_PO,
              oDriveStD_double_Param := "Station_MOVIKIT".MStNONE_PI,
              isCentering := #Centering_Perform[7, 1],
              HMI_StS_StD := "HMI_Pallets".Run_Command_right_ROW4[4],
              HMI_StD_StS := "HMI_Pallets".Run_Command_left_ROW4[4],
              oButton_StS_StD_LED => "Sz8_Button_LED_ST06_ST07",
              oStatus_HMI_StS_StD => "HMI_Pallets".Run_Status_right_ROW4[4],
              oStatus_HMI_StD_StS => "HMI_Pallets".Run_Status_left_ROW4[4],
              oCentering => #Centering_Status[7, 1],
              Stop_Drive_Button => "HMI_Pallets".Stop_Driver_Button1.%X6,
              Stop_Drive_HMI => "HMI_Pallets".Stop_Driver_HMI1.%X6);
END_REGION

REGION Network 59: ST05->ST06
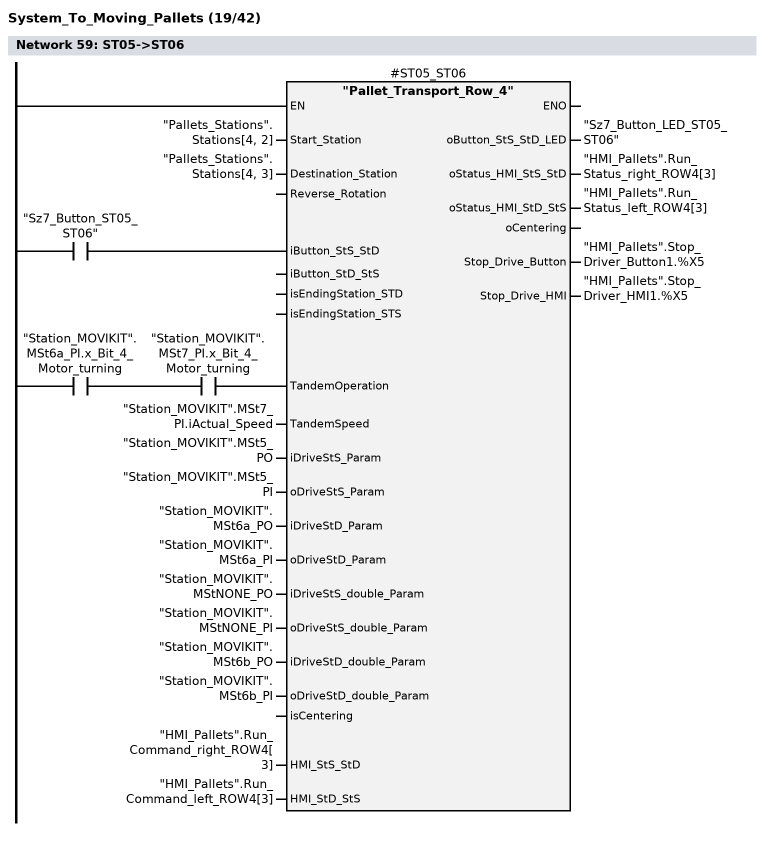
   RUNG wire#powerrail
      #ST05_ST06(iButton_StS_StD := wire#w1, TandemOperation := wire#w2, Start_Station := "Pallets_Stations".Stations[4, 2], Destination_Station := "Pallets_Stations".Stations[4, 3], Reverse_Rotation :=, iButton_StD_StS :=, isEndingStation_STD :=, isEndingStation_STS :=, TandemSpeed := "Station_MOVIKIT".MSt7_PI.iActual_Speed, iDriveStS_Param := "Station_MOVIKIT".MSt5_PO, oDriveStS_Param := "Station_MOVIKIT".MSt5_PI, iDriveStD_Param := "Station_MOVIKIT".MSt6a_PO, oDriveStD_Param := "Station_MOVIKIT".MSt6a_PI, iDriveStS_double_Param := "Station_MOVIKIT".MStNONE_PO, oDriveStS_double_Param := "Station_MOVIKIT".MStNONE_PI, iDriveStD_double_Param := "Station_MOVIKIT".MSt6b_PO, oDriveStD_double_Param := "Station_MOVIKIT".MSt6b_PI, isCentering :=, HMI_StS_StD := "HMI_Pallets".Run_Command_right_ROW4[3], HMI_StD_StS := "HMI_Pallets".Run_Command_left_ROW4[3], oButton_StS_StD_LED => "Sz7_Button_LED_ST05_ST06", oStatus_HMI_StS_StD => "HMI_Pallets".Run_Status_right_ROW4[3], oStatus_HMI_StD_StS => "HMI_Pallets".Run_Status_left_ROW4[3], oCentering =>, Stop_Drive_Button => "HMI_Pallets".Stop_Driver_Button1.%X5, Stop_Drive_HMI => "HMI_Pallets".Stop_Driver_HMI1.%X5)
   END_RUNG
   RUNG wire#powerrail
      Contact( "Sz7_Button_ST05_ST06" )
   END_RUNG wire#w1
   RUNG wire#powerrail
      Contact( "Station_MOVIKIT".MSt6a_PI.x_Bit_4_Motor_turning )
      Contact( "Station_MOVIKIT".MSt7_PI.x_Bit_4_Motor_turning )
   END_RUNG wire#w2
   // the same network as SCL:
   #ST05_ST06(Start_Station := "Pallets_Stations".Stations[4, 2],   // "Pallet_Transport_Row_4"
              Destination_Station := "Pallets_Stations".Stations[4, 3],
              iButton_StS_StD := "Sz7_Button_ST05_ST06",
              TandemOperation := "Station_MOVIKIT".MSt6a_PI.x_Bit_4_Motor_turning AND "Station_MOVIKIT".MSt7_PI.x_Bit_4_Motor_turning,
              TandemSpeed := "Station_MOVIKIT".MSt7_PI.iActual_Speed,
              iDriveStS_Param := "Station_MOVIKIT".MSt5_PO,
              oDriveStS_Param := "Station_MOVIKIT".MSt5_PI,
              iDriveStD_Param := "Station_MOVIKIT".MSt6a_PO,
              oDriveStD_Param := "Station_MOVIKIT".MSt6a_PI,
              iDriveStS_double_Param := "Station_MOVIKIT".MStNONE_PO,
              oDriveStS_double_Param := "Station_MOVIKIT".MStNONE_PI,
              iDriveStD_double_Param := "Station_MOVIKIT".MSt6b_PO,
              oDriveStD_double_Param := "Station_MOVIKIT".MSt6b_PI,
              HMI_StS_StD := "HMI_Pallets".Run_Command_right_ROW4[3],
              HMI_StD_StS := "HMI_Pallets".Run_Command_left_ROW4[3],
              oButton_StS_StD_LED => "Sz7_Button_LED_ST05_ST06",
              oStatus_HMI_StS_StD => "HMI_Pallets".Run_Status_right_ROW4[3],
              oStatus_HMI_StD_StS => "HMI_Pallets".Run_Status_left_ROW4[3],
              Stop_Drive_Button => "HMI_Pallets".Stop_Driver_Button1.%X5,
              Stop_Drive_HMI => "HMI_Pallets".Stop_Driver_HMI1.%X5);
END_REGION

REGION Network 60: ST04->ST05
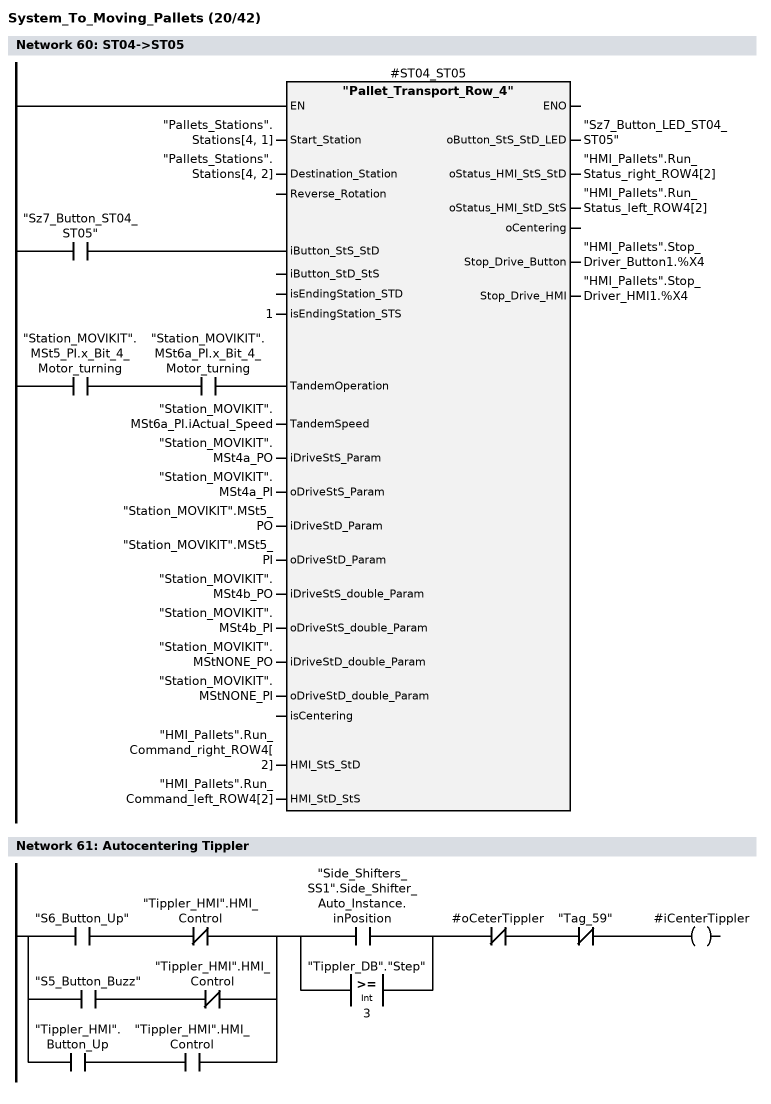
   RUNG wire#powerrail
      #ST04_ST05(iButton_StS_StD := wire#w1, TandemOperation := wire#w2, Start_Station := "Pallets_Stations".Stations[4, 1], Destination_Station := "Pallets_Stations".Stations[4, 2], Reverse_Rotation :=, iButton_StD_StS :=, isEndingStation_STD :=, isEndingStation_STS := 1, TandemSpeed := "Station_MOVIKIT".MSt6a_PI.iActual_Speed, iDriveStS_Param := "Station_MOVIKIT".MSt4a_PO, oDriveStS_Param := "Station_MOVIKIT".MSt4a_PI, iDriveStD_Param := "Station_MOVIKIT".MSt5_PO, oDriveStD_Param := "Station_MOVIKIT".MSt5_PI, iDriveStS_double_Param := "Station_MOVIKIT".MSt4b_PO, oDriveStS_double_Param := "Station_MOVIKIT".MSt4b_PI, iDriveStD_double_Param := "Station_MOVIKIT".MStNONE_PO, oDriveStD_double_Param := "Station_MOVIKIT".MStNONE_PI, isCentering :=, HMI_StS_StD := "HMI_Pallets".Run_Command_right_ROW4[2], HMI_StD_StS := "HMI_Pallets".Run_Command_left_ROW4[2], oButton_StS_StD_LED => "Sz7_Button_LED_ST04_ST05", oStatus_HMI_StS_StD => "HMI_Pallets".Run_Status_right_ROW4[2], oStatus_HMI_StD_StS => "HMI_Pallets".Run_Status_left_ROW4[2], oCentering =>, Stop_Drive_Button => "HMI_Pallets".Stop_Driver_Button1.%X4, Stop_Drive_HMI => "HMI_Pallets".Stop_Driver_HMI1.%X4)
   END_RUNG
   RUNG wire#powerrail
      Contact( "Sz7_Button_ST04_ST05" )
   END_RUNG wire#w1
   RUNG wire#powerrail
      Contact( "Station_MOVIKIT".MSt5_PI.x_Bit_4_Motor_turning )
      Contact( "Station_MOVIKIT".MSt6a_PI.x_Bit_4_Motor_turning )
   END_RUNG wire#w2
   // the same network as SCL:
   #ST04_ST05(Start_Station := "Pallets_Stations".Stations[4, 1],   // "Pallet_Transport_Row_4"
              Destination_Station := "Pallets_Stations".Stations[4, 2],
              iButton_StS_StD := "Sz7_Button_ST04_ST05",
              isEndingStation_STS := 1,
              TandemOperation := "Station_MOVIKIT".MSt5_PI.x_Bit_4_Motor_turning AND "Station_MOVIKIT".MSt6a_PI.x_Bit_4_Motor_turning,
              TandemSpeed := "Station_MOVIKIT".MSt6a_PI.iActual_Speed,
              iDriveStS_Param := "Station_MOVIKIT".MSt4a_PO,
              oDriveStS_Param := "Station_MOVIKIT".MSt4a_PI,
              iDriveStD_Param := "Station_MOVIKIT".MSt5_PO,
              oDriveStD_Param := "Station_MOVIKIT".MSt5_PI,
              iDriveStS_double_Param := "Station_MOVIKIT".MSt4b_PO,
              oDriveStS_double_Param := "Station_MOVIKIT".MSt4b_PI,
              iDriveStD_double_Param := "Station_MOVIKIT".MStNONE_PO,
              oDriveStD_double_Param := "Station_MOVIKIT".MStNONE_PI,
              HMI_StS_StD := "HMI_Pallets".Run_Command_right_ROW4[2],
              HMI_StD_StS := "HMI_Pallets".Run_Command_left_ROW4[2],
              oButton_StS_StD_LED => "Sz7_Button_LED_ST04_ST05",
              oStatus_HMI_StS_StD => "HMI_Pallets".Run_Status_right_ROW4[2],
              oStatus_HMI_StD_StS => "HMI_Pallets".Run_Status_left_ROW4[2],
              Stop_Drive_Button => "HMI_Pallets".Stop_Driver_Button1.%X4,
              Stop_Drive_HMI => "HMI_Pallets".Stop_Driver_HMI1.%X4);
END_REGION

REGION Network 61: Autocentering Tippler
   RUNG wire#powerrail
      Contact( "S6_Button_Up" )
      I_Contact( "Tippler_HMI".HMI_Control )
      wire#w1
      Contact( "Side_Shifters_SS1".Side_Shifter_Auto_Instance.inPosition )
      wire#w2
      I_Contact( #oCeterTippler )
      I_Contact( "Tag_59" )
      Coil( #iCenterTippler )
   END_RUNG
   RUNG wire#powerrail
      Contact( "S5_Button_Buzz" )
      I_Contact( "Tippler_HMI".HMI_Control )
   END_RUNG wire#w1
   RUNG wire#powerrail
      Contact( "Tippler_HMI".Button_Up )
      Contact( "Tippler_HMI".HMI_Control )
   END_RUNG wire#w1
   RUNG wire#w1
      { S7_Templates := "SrcType := Int" } GE_Contact(in1 := "Tippler_DB"."Step", in2 := 3)
   END_RUNG wire#w2
   // the same network as SCL:
   #iCenterTippler := (("S6_Button_Up" AND NOT "Tippler_HMI".HMI_Control) OR ("S5_Button_Buzz" AND NOT "Tippler_HMI".HMI_Control) OR ("Tippler_HMI".Button_Up AND "Tippler_HMI".HMI_Control)) AND ("Side_Shifters_SS1".Side_Shifter_Auto_Instance.inPosition OR ("Tippler_DB"."Step" >= 3)) AND NOT #oCeterTippler AND NOT "Tag_59";
END_REGION

REGION Network 62: ST01->ST02
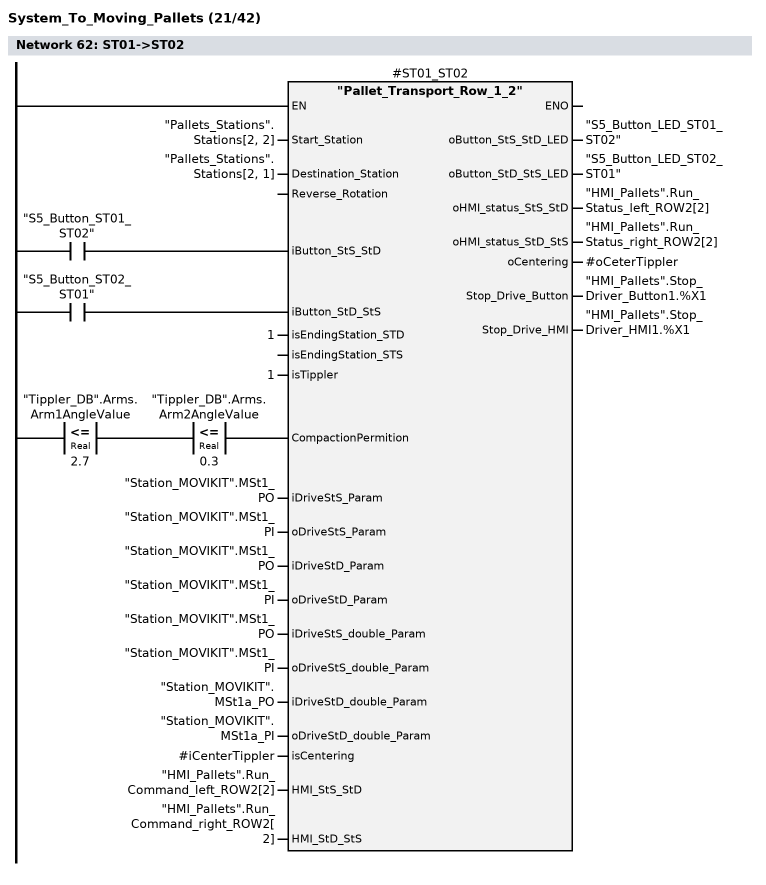
   RUNG wire#powerrail
      #ST01_ST02(iButton_StS_StD := wire#w1, iButton_StD_StS := wire#w2, CompactionPermition := wire#w3, Start_Station := "Pallets_Stations".Stations[2, 2], Destination_Station := "Pallets_Stations".Stations[2, 1], Reverse_Rotation :=, isEndingStation_STD := 1, isEndingStation_STS :=, isTippler := 1, iDriveStS_Param := "Station_MOVIKIT".MSt1_PO, oDriveStS_Param := "Station_MOVIKIT".MSt1_PI, iDriveStD_Param := "Station_MOVIKIT".MSt1_PO, oDriveStD_Param := "Station_MOVIKIT".MSt1_PI, iDriveStS_double_Param := "Station_MOVIKIT".MSt1_PO, oDriveStS_double_Param := "Station_MOVIKIT".MSt1_PI, iDriveStD_double_Param := "Station_MOVIKIT".MSt1a_PO, oDriveStD_double_Param := "Station_MOVIKIT".MSt1a_PI, isCentering := #iCenterTippler, HMI_StS_StD := "HMI_Pallets".Run_Command_left_ROW2[2], HMI_StD_StS := "HMI_Pallets".Run_Command_right_ROW2[2], oButton_StS_StD_LED => "S5_Button_LED_ST01_ST02", oButton_StD_StS_LED => "S5_Button_LED_ST02_ST01", oHMI_status_StS_StD => "HMI_Pallets".Run_Status_left_ROW2[2], oHMI_status_StD_StS => "HMI_Pallets".Run_Status_right_ROW2[2], oCentering => #oCeterTippler, Stop_Drive_Button => "HMI_Pallets".Stop_Driver_Button1.%X1, Stop_Drive_HMI => "HMI_Pallets".Stop_Driver_HMI1.%X1)
   END_RUNG
   RUNG wire#powerrail
      Contact( "S5_Button_ST01_ST02" )
   END_RUNG wire#w1
   RUNG wire#powerrail
      Contact( "S5_Button_ST02_ST01" )
   END_RUNG wire#w2
   RUNG wire#powerrail
      { S7_Templates := "SrcType := Real" } LE_Contact(in1 := "Tippler_DB".Arms.Arm1AngleValue, in2 := 2.7)
      { S7_Templates := "SrcType := Real" } LE_Contact(in1 := "Tippler_DB".Arms.Arm2AngleValue, in2 := 0.3)
   END_RUNG wire#w3
   // the same network as SCL:
   #ST01_ST02(Start_Station := "Pallets_Stations".Stations[2, 2],   // "Pallet_Transport_Row_1_2"
              Destination_Station := "Pallets_Stations".Stations[2, 1],
              iButton_StS_StD := "S5_Button_ST01_ST02",
              iButton_StD_StS := "S5_Button_ST02_ST01",
              isEndingStation_STD := 1,
              isTippler := 1,
              CompactionPermition := ("Tippler_DB".Arms.Arm1AngleValue <= 2.7) AND ("Tippler_DB".Arms.Arm2AngleValue <= 0.3),
              iDriveStS_Param := "Station_MOVIKIT".MSt1_PO,
              oDriveStS_Param := "Station_MOVIKIT".MSt1_PI,
              iDriveStD_Param := "Station_MOVIKIT".MSt1_PO,
              oDriveStD_Param := "Station_MOVIKIT".MSt1_PI,
              iDriveStS_double_Param := "Station_MOVIKIT".MSt1_PO,
              oDriveStS_double_Param := "Station_MOVIKIT".MSt1_PI,
              iDriveStD_double_Param := "Station_MOVIKIT".MSt1a_PO,
              oDriveStD_double_Param := "Station_MOVIKIT".MSt1a_PI,
              isCentering := #iCenterTippler,
              HMI_StS_StD := "HMI_Pallets".Run_Command_left_ROW2[2],
              HMI_StD_StS := "HMI_Pallets".Run_Command_right_ROW2[2],
              oButton_StS_StD_LED => "S5_Button_LED_ST01_ST02",
              oButton_StD_StS_LED => "S5_Button_LED_ST02_ST01",
              oHMI_status_StS_StD => "HMI_Pallets".Run_Status_left_ROW2[2],
              oHMI_status_StD_StS => "HMI_Pallets".Run_Status_right_ROW2[2],
              oCentering => #oCeterTippler,
              Stop_Drive_Button => "HMI_Pallets".Stop_Driver_Button1.%X1,
              Stop_Drive_HMI => "HMI_Pallets".Stop_Driver_HMI1.%X1);
END_REGION

REGION Network 63: ST38->ST01
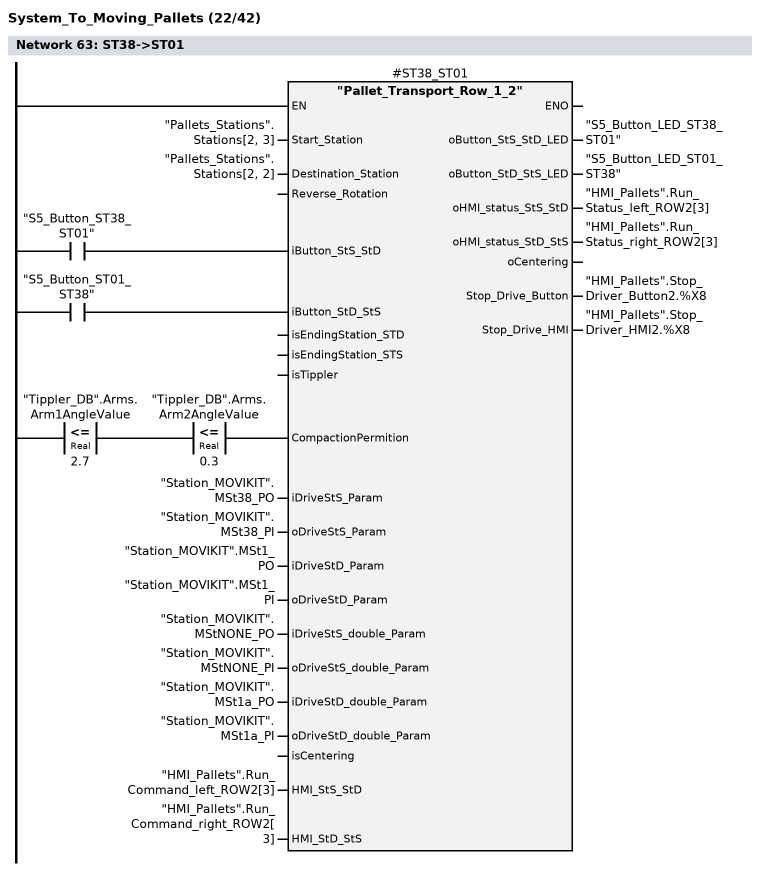
   RUNG wire#powerrail
      #ST38_ST01(iButton_StS_StD := wire#w1, iButton_StD_StS := wire#w2, CompactionPermition := wire#w3, Start_Station := "Pallets_Stations".Stations[2, 3], Destination_Station := "Pallets_Stations".Stations[2, 2], Reverse_Rotation :=, isEndingStation_STD :=, isEndingStation_STS :=, isTippler :=, iDriveStS_Param := "Station_MOVIKIT".MSt38_PO, oDriveStS_Param := "Station_MOVIKIT".MSt38_PI, iDriveStD_Param := "Station_MOVIKIT".MSt1_PO, oDriveStD_Param := "Station_MOVIKIT".MSt1_PI, iDriveStS_double_Param := "Station_MOVIKIT".MStNONE_PO, oDriveStS_double_Param := "Station_MOVIKIT".MStNONE_PI, iDriveStD_double_Param := "Station_MOVIKIT".MSt1a_PO, oDriveStD_double_Param := "Station_MOVIKIT".MSt1a_PI, isCentering :=, HMI_StS_StD := "HMI_Pallets".Run_Command_left_ROW2[3], HMI_StD_StS := "HMI_Pallets".Run_Command_right_ROW2[3], oButton_StS_StD_LED => "S5_Button_LED_ST38_ST01", oButton_StD_StS_LED => "S5_Button_LED_ST01_ST38", oHMI_status_StS_StD => "HMI_Pallets".Run_Status_left_ROW2[3], oHMI_status_StD_StS => "HMI_Pallets".Run_Status_right_ROW2[3], oCentering =>, Stop_Drive_Button => "HMI_Pallets".Stop_Driver_Button2.%X8, Stop_Drive_HMI => "HMI_Pallets".Stop_Driver_HMI2.%X8)
   END_RUNG
   RUNG wire#powerrail
      Contact( "S5_Button_ST38_ST01" )
   END_RUNG wire#w1
   RUNG wire#powerrail
      Contact( "S5_Button_ST01_ST38" )
   END_RUNG wire#w2
   RUNG wire#powerrail
      { S7_Templates := "SrcType := Real" } LE_Contact(in1 := "Tippler_DB".Arms.Arm1AngleValue, in2 := 2.7)
      { S7_Templates := "SrcType := Real" } LE_Contact(in1 := "Tippler_DB".Arms.Arm2AngleValue, in2 := 0.3)
   END_RUNG wire#w3
   // the same network as SCL:
   #ST38_ST01(Start_Station := "Pallets_Stations".Stations[2, 3],   // "Pallet_Transport_Row_1_2"
              Destination_Station := "Pallets_Stations".Stations[2, 2],
              iButton_StS_StD := "S5_Button_ST38_ST01",
              iButton_StD_StS := "S5_Button_ST01_ST38",
              CompactionPermition := ("Tippler_DB".Arms.Arm1AngleValue <= 2.7) AND ("Tippler_DB".Arms.Arm2AngleValue <= 0.3),
              iDriveStS_Param := "Station_MOVIKIT".MSt38_PO,
              oDriveStS_Param := "Station_MOVIKIT".MSt38_PI,
              iDriveStD_Param := "Station_MOVIKIT".MSt1_PO,
              oDriveStD_Param := "Station_MOVIKIT".MSt1_PI,
              iDriveStS_double_Param := "Station_MOVIKIT".MStNONE_PO,
              oDriveStS_double_Param := "Station_MOVIKIT".MStNONE_PI,
              iDriveStD_double_Param := "Station_MOVIKIT".MSt1a_PO,
              oDriveStD_double_Param := "Station_MOVIKIT".MSt1a_PI,
              HMI_StS_StD := "HMI_Pallets".Run_Command_left_ROW2[3],
              HMI_StD_StS := "HMI_Pallets".Run_Command_right_ROW2[3],
              oButton_StS_StD_LED => "S5_Button_LED_ST38_ST01",
              oButton_StD_StS_LED => "S5_Button_LED_ST01_ST38",
              oHMI_status_StS_StD => "HMI_Pallets".Run_Status_left_ROW2[3],
              oHMI_status_StD_StS => "HMI_Pallets".Run_Status_right_ROW2[3],
              Stop_Drive_Button => "HMI_Pallets".Stop_Driver_Button2.%X8,
              Stop_Drive_HMI => "HMI_Pallets".Stop_Driver_HMI2.%X8);
END_REGION

REGION Network 64: ST34->ST35
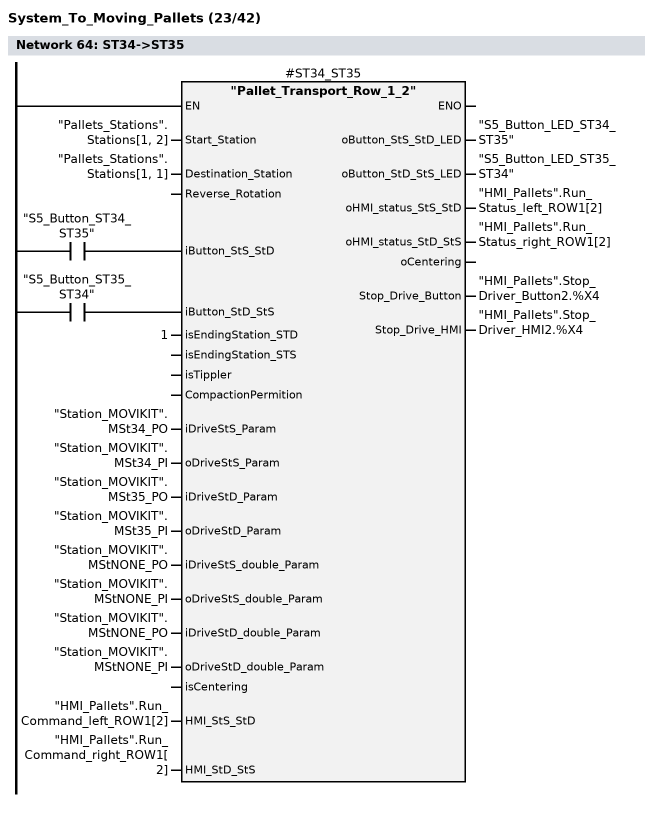
   RUNG wire#powerrail
      #ST34_ST35(iButton_StS_StD := wire#w1, iButton_StD_StS := wire#w2, Start_Station := "Pallets_Stations".Stations[1, 2], Destination_Station := "Pallets_Stations".Stations[1, 1], Reverse_Rotation :=, isEndingStation_STD := 1, isEndingStation_STS :=, isTippler :=, CompactionPermition :=, iDriveStS_Param := "Station_MOVIKIT".MSt34_PO, oDriveStS_Param := "Station_MOVIKIT".MSt34_PI, iDriveStD_Param := "Station_MOVIKIT".MSt35_PO, oDriveStD_Param := "Station_MOVIKIT".MSt35_PI, iDriveStS_double_Param := "Station_MOVIKIT".MStNONE_PO, oDriveStS_double_Param := "Station_MOVIKIT".MStNONE_PI, iDriveStD_double_Param := "Station_MOVIKIT".MStNONE_PO, oDriveStD_double_Param := "Station_MOVIKIT".MStNONE_PI, isCentering :=, HMI_StS_StD := "HMI_Pallets".Run_Command_left_ROW1[2], HMI_StD_StS := "HMI_Pallets".Run_Command_right_ROW1[2], oButton_StS_StD_LED => "S5_Button_LED_ST34_ST35", oButton_StD_StS_LED => "S5_Button_LED_ST35_ST34", oHMI_status_StS_StD => "HMI_Pallets".Run_Status_left_ROW1[2], oHMI_status_StD_StS => "HMI_Pallets".Run_Status_right_ROW1[2], oCentering =>, Stop_Drive_Button => "HMI_Pallets".Stop_Driver_Button2.%X4, Stop_Drive_HMI => "HMI_Pallets".Stop_Driver_HMI2.%X4)
   END_RUNG
   RUNG wire#powerrail
      Contact( "S5_Button_ST34_ST35" )
   END_RUNG wire#w1
   RUNG wire#powerrail
      Contact( "S5_Button_ST35_ST34" )
   END_RUNG wire#w2
   // the same network as SCL:
   #ST34_ST35(Start_Station := "Pallets_Stations".Stations[1, 2],   // "Pallet_Transport_Row_1_2"
              Destination_Station := "Pallets_Stations".Stations[1, 1],
              iButton_StS_StD := "S5_Button_ST34_ST35",
              iButton_StD_StS := "S5_Button_ST35_ST34",
              isEndingStation_STD := 1,
              iDriveStS_Param := "Station_MOVIKIT".MSt34_PO,
              oDriveStS_Param := "Station_MOVIKIT".MSt34_PI,
              iDriveStD_Param := "Station_MOVIKIT".MSt35_PO,
              oDriveStD_Param := "Station_MOVIKIT".MSt35_PI,
              iDriveStS_double_Param := "Station_MOVIKIT".MStNONE_PO,
              oDriveStS_double_Param := "Station_MOVIKIT".MStNONE_PI,
              iDriveStD_double_Param := "Station_MOVIKIT".MStNONE_PO,
              oDriveStD_double_Param := "Station_MOVIKIT".MStNONE_PI,
              HMI_StS_StD := "HMI_Pallets".Run_Command_left_ROW1[2],
              HMI_StD_StS := "HMI_Pallets".Run_Command_right_ROW1[2],
              oButton_StS_StD_LED => "S5_Button_LED_ST34_ST35",
              oButton_StD_StS_LED => "S5_Button_LED_ST35_ST34",
              oHMI_status_StS_StD => "HMI_Pallets".Run_Status_left_ROW1[2],
              oHMI_status_StD_StS => "HMI_Pallets".Run_Status_right_ROW1[2],
              Stop_Drive_Button => "HMI_Pallets".Stop_Driver_Button2.%X4,
              Stop_Drive_HMI => "HMI_Pallets".Stop_Driver_HMI2.%X4);
END_REGION

REGION Network 65: ST33->ST34
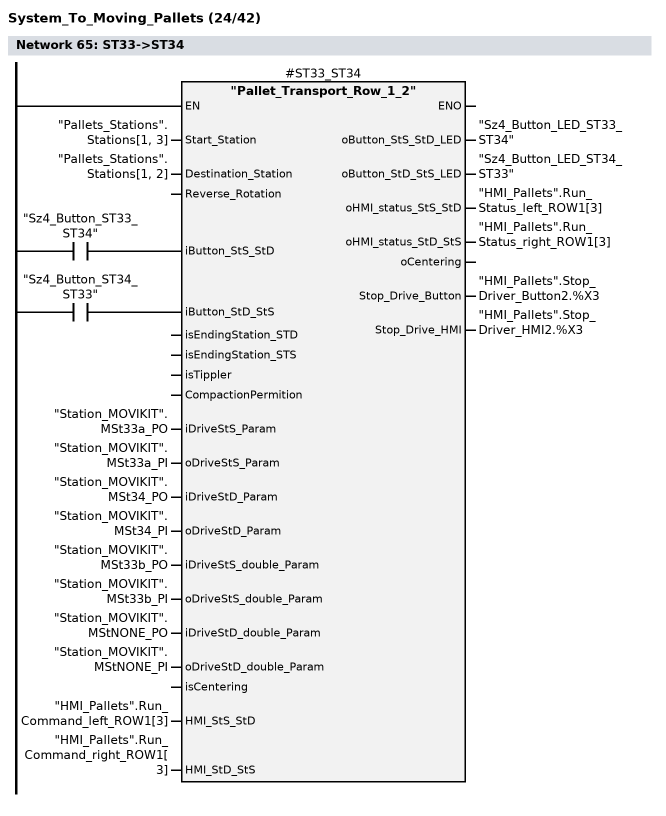
   RUNG wire#powerrail
      #ST33_ST34(iButton_StS_StD := wire#w1, iButton_StD_StS := wire#w2, Start_Station := "Pallets_Stations".Stations[1, 3], Destination_Station := "Pallets_Stations".Stations[1, 2], Reverse_Rotation :=, isEndingStation_STD :=, isEndingStation_STS :=, isTippler :=, CompactionPermition :=, iDriveStS_Param := "Station_MOVIKIT".MSt33a_PO, oDriveStS_Param := "Station_MOVIKIT".MSt33a_PI, iDriveStD_Param := "Station_MOVIKIT".MSt34_PO, oDriveStD_Param := "Station_MOVIKIT".MSt34_PI, iDriveStS_double_Param := "Station_MOVIKIT".MSt33b_PO, oDriveStS_double_Param := "Station_MOVIKIT".MSt33b_PI, iDriveStD_double_Param := "Station_MOVIKIT".MStNONE_PO, oDriveStD_double_Param := "Station_MOVIKIT".MStNONE_PI, isCentering :=, HMI_StS_StD := "HMI_Pallets".Run_Command_left_ROW1[3], HMI_StD_StS := "HMI_Pallets".Run_Command_right_ROW1[3], oButton_StS_StD_LED => "Sz4_Button_LED_ST33_ST34", oButton_StD_StS_LED => "Sz4_Button_LED_ST34_ST33", oHMI_status_StS_StD => "HMI_Pallets".Run_Status_left_ROW1[3], oHMI_status_StD_StS => "HMI_Pallets".Run_Status_right_ROW1[3], oCentering =>, Stop_Drive_Button => "HMI_Pallets".Stop_Driver_Button2.%X3, Stop_Drive_HMI => "HMI_Pallets".Stop_Driver_HMI2.%X3)
   END_RUNG
   RUNG wire#powerrail
      Contact( "Sz4_Button_ST33_ST34" )
   END_RUNG wire#w1
   RUNG wire#powerrail
      Contact( "Sz4_Button_ST34_ST33" )
   END_RUNG wire#w2
   // the same network as SCL:
   #ST33_ST34(Start_Station := "Pallets_Stations".Stations[1, 3],   // "Pallet_Transport_Row_1_2"
              Destination_Station := "Pallets_Stations".Stations[1, 2],
              iButton_StS_StD := "Sz4_Button_ST33_ST34",
              iButton_StD_StS := "Sz4_Button_ST34_ST33",
              iDriveStS_Param := "Station_MOVIKIT".MSt33a_PO,
              oDriveStS_Param := "Station_MOVIKIT".MSt33a_PI,
              iDriveStD_Param := "Station_MOVIKIT".MSt34_PO,
              oDriveStD_Param := "Station_MOVIKIT".MSt34_PI,
              iDriveStS_double_Param := "Station_MOVIKIT".MSt33b_PO,
              oDriveStS_double_Param := "Station_MOVIKIT".MSt33b_PI,
              iDriveStD_double_Param := "Station_MOVIKIT".MStNONE_PO,
              oDriveStD_double_Param := "Station_MOVIKIT".MStNONE_PI,
              HMI_StS_StD := "HMI_Pallets".Run_Command_left_ROW1[3],
              HMI_StD_StS := "HMI_Pallets".Run_Command_right_ROW1[3],
              oButton_StS_StD_LED => "Sz4_Button_LED_ST33_ST34",
              oButton_StD_StS_LED => "Sz4_Button_LED_ST34_ST33",
              oHMI_status_StS_StD => "HMI_Pallets".Run_Status_left_ROW1[3],
              oHMI_status_StD_StS => "HMI_Pallets".Run_Status_right_ROW1[3],
              Stop_Drive_Button => "HMI_Pallets".Stop_Driver_Button2.%X3,
              Stop_Drive_HMI => "HMI_Pallets".Stop_Driver_HMI2.%X3);
END_REGION

REGION Network 66: ST32->ST33
